DATA_BLOCK "_2010SC130U01TSH01_DB"   // DB2038
TITLE = Instance DB Alarm: Break Resistor Temp High
{ S7_Optimized_Access := 'FALSE' }
AUTHOR : 7Art
NAME : ALARM_DB
VERSION : 8.0
// stored: InstanceOfName ACESYS_ALARM
"ACESYS_ALARM"
BEGIN
   FP_PARM.EnableTime_Low_Pre := 5;
   FP_EN.Alarm_Low := TRUE;
   PWR := TRUE;
   EN_L := TRUE;
   OK := TRUE;
   AL_L := TRUE;
   AL_H := TRUE;
   WARN_L := TRUE;
   WARN_H := TRUE;
   MSW.EXT.Operation := TRUE;
   MSW.Status := 2;
   MSW.TimeStamp := 16#7ECD;
   BlockInfo.Ace_Version := 80;
   BlockInfo.Ace_BuildNo := 4;
   BlockInfo.State_Act := 2;
   BlockInfo.State_Prev := 202;
   BlockInfo.DB_Number := 2038;
   FP_PARM.EnableTime_Low_Acc := 5;
   FP_SIM.SIG_Enable := TRUE;
   FP_SIM.PWR_Enable := TRUE;
   ONS.SecPulse1 := TRUE;
   ONS.AL_L_Aux := TRUE;
   ONS.AL_H_Aux := TRUE;
   EnableTime_Low_Done := TRUE;
   StatusWork := 2;
   OUT.OK := TRUE;
   OUT.AL_L := TRUE;
   OUT.AL_H := TRUE;
   OUT.WARN_L := TRUE;
   OUT.WARN_H := TRUE;
   MSW_Status_Trans := 2;
END_DATA_BLOCK

DATA_BLOCK "_2010CR150M01OAC01_DB"   // DB2039
TITLE = Instance DB Alarm: Emergency stop PB
{ S7_Optimized_Access := 'FALSE' }
AUTHOR : 7Art
NAME : ALARM_DB
VERSION : 8.0
// stored: InstanceOfName ACESYS_ALARM
"ACESYS_ALARM"
BEGIN
   FP_PARM.EnableTime_Low_Pre := 5;
   FP_EN.Alarm_Low := TRUE;
   PWR := TRUE;
   EN_L := TRUE;
   OK := TRUE;
   AL_L := TRUE;
   AL_H := TRUE;
   WARN_L := TRUE;
   WARN_H := TRUE;
   MSW.EXT.Operation := TRUE;
   MSW.Status := 2;
   MSW.TimeStamp := 16#72EA;
   BlockInfo.Ace_Version := 80;
   BlockInfo.Ace_BuildNo := 4;
   BlockInfo.State_Act := 2;
   BlockInfo.State_Prev := 202;
   BlockInfo.DB_Number := 2039;
   FP_PARM.EnableTime_Low_Acc := 5;
   FP_SIM.SIG_Enable := TRUE;
   FP_SIM.PWR_Enable := TRUE;
   ONS.SecPulse1 := TRUE;
   ONS.AL_L_Aux := TRUE;
   ONS.AL_H_Aux := TRUE;
   EnableTime_Low_Done := TRUE;
   StatusWork := 2;
   OUT.OK := TRUE;
   OUT.AL_L := TRUE;
   OUT.AL_H := TRUE;
   OUT.WARN_L := TRUE;
   OUT.WARN_H := TRUE;
   MSW_Status_Trans := 2;
END_DATA_BLOCK

DATA_BLOCK "_2010CR150M01YSQ01_DB"   // DB2040
TITLE = Instance DB Alarm: Breaker feedback
{ S7_Optimized_Access := 'FALSE' }
AUTHOR : 7Art
NAME : ALARM_DB
VERSION : 8.0
// stored: InstanceOfName ACESYS_ALARM
"ACESYS_ALARM"
BEGIN
   FP_PARM.EnableTime_Low_Pre := 5;
   FP_EN.Alarm_Low := TRUE;
   PWR := TRUE;
   EN_L := TRUE;
   OK := TRUE;
   AL_L := TRUE;
   AL_H := TRUE;
   WARN_L := TRUE;
   WARN_H := TRUE;
   MSW.EXT.Operation := TRUE;
   MSW.Status := 2;
   MSW.TimeStamp := 16#8D11;
   BlockInfo.Ace_Version := 80;
   BlockInfo.Ace_BuildNo := 4;
   BlockInfo.State_Act := 2;
   BlockInfo.State_Prev := 202;
   BlockInfo.DB_Number := 2040;
   FP_PARM.EnableTime_Low_Acc := 5;
   FP_SIM.SIG_Enable := TRUE;
   FP_SIM.PWR_Enable := TRUE;
   ONS.SecPulse1 := TRUE;
   ONS.AL_L_Aux := TRUE;
   ONS.AL_H_Aux := TRUE;
   EnableTime_Low_Done := TRUE;
   StatusWork := 2;
   OUT.OK := TRUE;
   OUT.AL_L := TRUE;
   OUT.AL_H := TRUE;
   OUT.WARN_L := TRUE;
   OUT.WARN_H := TRUE;
   MSW_Status_Trans := 2;
END_DATA_BLOCK

DATA_BLOCK "_2010CR150M01NS01_DB"   // DB2041
TITLE = Instance DB Alarm: PTS Sensor
{ S7_Optimized_Access := 'FALSE' }
AUTHOR : 7Art
NAME : ALARM_DB
VERSION : 8.0
// stored: InstanceOfName ACESYS_ALARM
"ACESYS_ALARM"
BEGIN
   FP_PARM.EnableTime_Low_Pre := 5;
   FP_EN.Alarm_Low := TRUE;
   PWR := TRUE;
   EN_L := TRUE;
   OK := TRUE;
   AL_L := TRUE;
   AL_H := TRUE;
   WARN_L := TRUE;
   WARN_H := TRUE;
   MSW.EXT.Operation := TRUE;
   MSW.Status := 2;
   MSW.TimeStamp := 16#08E4;
   BlockInfo.Ace_Version := 80;
   BlockInfo.Ace_BuildNo := 4;
   BlockInfo.State_Act := 2;
   BlockInfo.State_Prev := 202;
   BlockInfo.DB_Number := 2041;
   FP_PARM.EnableTime_Low_Acc := 5;
   FP_SIM.SIG_Enable := TRUE;
   FP_SIM.PWR_Enable := TRUE;
   ONS.SecPulse1 := TRUE;
   ONS.AL_L_Aux := TRUE;
   ONS.AL_H_Aux := TRUE;
   EnableTime_Low_Done := TRUE;
   StatusWork := 2;
   OUT.OK := TRUE;
   OUT.AL_L := TRUE;
   OUT.AL_H := TRUE;
   OUT.WARN_L := TRUE;
   OUT.WARN_H := TRUE;
   MSW_Status_Trans := 2;
END_DATA_BLOCK

DATA_BLOCK "_2010PMC01YSH01_DB"   // DB2042
TITLE = Instance DB Alarm: PTS Sensor
{ S7_Optimized_Access := 'FALSE' }
AUTHOR : 7Art
NAME : ALARM_DB
VERSION : 8.0
// stored: InstanceOfName ACESYS_ALARM
"ACESYS_ALARM"
BEGIN
   FP_PARM.EnableTime_Low_Pre := 5;
   FP_EN.Alarm_Low := TRUE;
   PWR := TRUE;
   EN_L := TRUE;
   OK := TRUE;
   AL_L := TRUE;
   AL_H := TRUE;
   WARN_L := TRUE;
   WARN_H := TRUE;
   MSW.EXT.Operation := TRUE;
   MSW.Status := 2;
   MSW.TimeStamp := 16#8C12;
   BlockInfo.Ace_Version := 80;
   BlockInfo.Ace_BuildNo := 4;
   BlockInfo.State_Act := 2;
   BlockInfo.State_Prev := 202;
   BlockInfo.DB_Number := 2042;
   FP_PARM.EnableTime_Low_Acc := 5;
   FP_SIM.SIG_Enable := TRUE;
   FP_SIM.PWR_Enable := TRUE;
   ONS.SecPulse1 := TRUE;
   ONS.AL_L_Aux := TRUE;
   ONS.AL_H_Aux := TRUE;
   EnableTime_Low_Done := TRUE;
   StatusWork := 2;
   OUT.OK := TRUE;
   OUT.AL_L := TRUE;
   OUT.AL_H := TRUE;
   OUT.WARN_L := TRUE;
   OUT.WARN_H := TRUE;
   MSW_Status_Trans := 2;
END_DATA_BLOCK

DATA_BLOCK "_2010PMC01YSQ10G01_DB"   // DB2043
TITLE = Instance DB Alarm: PTS Sensor
{ S7_Optimized_Access := 'FALSE' }
AUTHOR : 7Art
NAME : ALARM_DB
VERSION : 8.0
// stored: InstanceOfName ACESYS_ALARM
"ACESYS_ALARM"
BEGIN
   FP_PARM.EnableTime_Low_Pre := 5;
   FP_EN.Alarm_Low := TRUE;
   PWR := TRUE;
   EN_L := TRUE;
   OK := TRUE;
   AL_L := TRUE;
   AL_H := TRUE;
   WARN_L := TRUE;
   WARN_H := TRUE;
   MSW.EXT.Operation := TRUE;
   MSW.Status := 2;
   MSW.TimeStamp := 16#8BF2;
   BlockInfo.Ace_Version := 80;
   BlockInfo.Ace_BuildNo := 4;
   BlockInfo.State_Act := 2;
   BlockInfo.State_Prev := 202;
   BlockInfo.DB_Number := 2043;
   FP_PARM.EnableTime_Low_Acc := 5;
   FP_SIM.SIG_Enable := TRUE;
   FP_SIM.PWR_Enable := TRUE;
   ONS.SecPulse2 := TRUE;
   ONS.AL_L_Aux := TRUE;
   ONS.AL_H_Aux := TRUE;
   EnableTime_Low_Done := TRUE;
   Sec_Pulse := TRUE;
   StatusWork := 2;
   OUT.OK := TRUE;
   OUT.AL_L := TRUE;
   OUT.AL_H := TRUE;
   OUT.WARN_L := TRUE;
   OUT.WARN_H := TRUE;
   MSW_Status_Trans := 2;
END_DATA_BLOCK

DATA_BLOCK "_2010PMC01YSQ10Q03_DB"   // DB2044
TITLE = Instance DB Alarm: PTS Sensor
{ S7_Optimized_Access := 'FALSE' }
AUTHOR : 7Art
NAME : ALARM_DB
VERSION : 8.0
// stored: InstanceOfName ACESYS_ALARM
"ACESYS_ALARM"
BEGIN
   FP_PARM.EnableTime_Low_Pre := 5;
   FP_EN.Alarm_Low := TRUE;
   PWR := TRUE;
   EN_L := TRUE;
   OK := TRUE;
   AL_L := TRUE;
   AL_H := TRUE;
   WARN_L := TRUE;
   WARN_H := TRUE;
   MSW.EXT.Operation := TRUE;
   MSW.Status := 2;
   MSW.TimeStamp := 16#7EC5;
   BlockInfo.Ace_Version := 80;
   BlockInfo.Ace_BuildNo := 4;
   BlockInfo.State_Act := 2;
   BlockInfo.State_Prev := 202;
   BlockInfo.DB_Number := 2044;
   FP_PARM.EnableTime_Low_Acc := 5;
   FP_SIM.SIG_Enable := TRUE;
   FP_SIM.PWR_Enable := TRUE;
   ONS.SecPulse2 := TRUE;
   ONS.AL_L_Aux := TRUE;
   ONS.AL_H_Aux := TRUE;
   EnableTime_Low_Done := TRUE;
   Sec_Pulse := TRUE;
   StatusWork := 2;
   OUT.OK := TRUE;
   OUT.AL_L := TRUE;
   OUT.AL_H := TRUE;
   OUT.WARN_L := TRUE;
   OUT.WARN_H := TRUE;
   MSW_Status_Trans := 2;
END_DATA_BLOCK

DATA_BLOCK "_2010PMC01YSQ20Q03_DB"   // DB2045
TITLE = Instance DB Alarm: PTS Sensor
{ S7_Optimized_Access := 'FALSE' }
AUTHOR : 7Art
NAME : ALARM_DB
VERSION : 8.0
// stored: InstanceOfName ACESYS_ALARM
"ACESYS_ALARM"
BEGIN
   FP_PARM.EnableTime_Low_Pre := 5;
   FP_EN.Alarm_Low := TRUE;
   PWR := TRUE;
   EN_L := TRUE;
   OK := TRUE;
   AL_L := TRUE;
   AL_H := TRUE;
   WARN_L := TRUE;
   WARN_H := TRUE;
   MSW.EXT.Operation := TRUE;
   MSW.Status := 2;
   MSW.TimeStamp := 16#72EA;
   BlockInfo.Ace_Version := 80;
   BlockInfo.Ace_BuildNo := 4;
   BlockInfo.State_Act := 2;
   BlockInfo.State_Prev := 202;
   BlockInfo.DB_Number := 2045;
   FP_PARM.EnableTime_Low_Acc := 5;
   FP_SIM.SIG_Enable := TRUE;
   FP_SIM.PWR_Enable := TRUE;
   ONS.SecPulse2 := TRUE;
   ONS.AL_L_Aux := TRUE;
   ONS.AL_H_Aux := TRUE;
   EnableTime_Low_Done := TRUE;
   StatusWork := 2;
   OUT.OK := TRUE;
   OUT.AL_L := TRUE;
   OUT.AL_H := TRUE;
   OUT.WARN_L := TRUE;
   OUT.WARN_H := TRUE;
   MSW_Status_Trans := 2;
END_DATA_BLOCK

DATA_BLOCK "_2010PMC01YSQ20Q04_DB"   // DB2046
TITLE = Instance DB Alarm: PTS Sensor
{ S7_Optimized_Access := 'FALSE' }
AUTHOR : 7Art
NAME : ALARM_DB
VERSION : 8.0
// stored: InstanceOfName ACESYS_ALARM
"ACESYS_ALARM"
BEGIN
   FP_PARM.EnableTime_Low_Pre := 5;
   FP_EN.Alarm_Low := TRUE;
   PWR := TRUE;
   EN_L := TRUE;
   OK := TRUE;
   AL_L := TRUE;
   AL_H := TRUE;
   WARN_L := TRUE;
   WARN_H := TRUE;
   MSW.EXT.Operation := TRUE;
   MSW.Status := 2;
   MSW.TimeStamp := 16#72EA;
   BlockInfo.Ace_Version := 80;
   BlockInfo.Ace_BuildNo := 4;
   BlockInfo.State_Act := 2;
   BlockInfo.State_Prev := 202;
   BlockInfo.DB_Number := 2046;
   FP_PARM.EnableTime_Low_Acc := 5;
   FP_SIM.SIG_Enable := TRUE;
   FP_SIM.PWR_Enable := TRUE;
   ONS.SecPulse2 := TRUE;
   ONS.AL_L_Aux := TRUE;
   ONS.AL_H_Aux := TRUE;
   EnableTime_Low_Done := TRUE;
   StatusWork := 2;
   OUT.OK := TRUE;
   OUT.AL_L := TRUE;
   OUT.AL_H := TRUE;
   OUT.WARN_L := TRUE;
   OUT.WARN_H := TRUE;
   MSW_Status_Trans := 2;
END_DATA_BLOCK

DATA_BLOCK "_2010PMC01YSQ26Q01_DB"   // DB2047
TITLE = Instance DB Alarm: PTS Sensor
{ S7_Optimized_Access := 'FALSE' }
AUTHOR : 7Art
NAME : ALARM_DB
VERSION : 8.0
// stored: InstanceOfName ACESYS_ALARM
"ACESYS_ALARM"
BEGIN
   FP_PARM.EnableTime_Low_Pre := 5;
   FP_EN.Alarm_Low := TRUE;
   PWR := TRUE;
   EN_L := TRUE;
   OK := TRUE;
   AL_L := TRUE;
   AL_H := TRUE;
   WARN_L := TRUE;
   WARN_H := TRUE;
   MSW.EXT.Operation := TRUE;
   MSW.Status := 2;
   MSW.TimeStamp := 16#61B4;
   BlockInfo.Ace_Version := 80;
   BlockInfo.Ace_BuildNo := 4;
   BlockInfo.State_Act := 2;
   BlockInfo.State_Prev := 202;
   BlockInfo.DB_Number := 2047;
   FP_PARM.EnableTime_Low_Acc := 5;
   FP_SIM.SIG_Enable := TRUE;
   FP_SIM.PWR_Enable := TRUE;
   ONS.SecPulse2 := TRUE;
   ONS.AL_L_Aux := TRUE;
   ONS.AL_H_Aux := TRUE;
   EnableTime_Low_Done := TRUE;
   StatusWork := 2;
   OUT.OK := TRUE;
   OUT.AL_L := TRUE;
   OUT.AL_H := TRUE;
   OUT.WARN_L := TRUE;
   OUT.WARN_H := TRUE;
   MSW_Status_Trans := 2;
END_DATA_BLOCK

DATA_BLOCK "_2010PMC01YSQ30Q02_DB"   // DB2048
TITLE = Instance DB Alarm: PTS Sensor
{ S7_Optimized_Access := 'FALSE' }
AUTHOR : 7Art
NAME : ALARM_DB
VERSION : 8.0
// stored: InstanceOfName ACESYS_ALARM
"ACESYS_ALARM"
BEGIN
   FP_PARM.EnableTime_Low_Pre := 5;
   FP_EN.Alarm_Low := TRUE;
   PWR := TRUE;
   EN_L := TRUE;
   OK := TRUE;
   AL_L := TRUE;
   AL_H := TRUE;
   WARN_L := TRUE;
   WARN_H := TRUE;
   MSW.EXT.Operation := TRUE;
   MSW.EXT.Forced := TRUE;
   MSW.Status := 2;
   MSW.TimeStamp := 16#166B;
   BlockInfo.Ace_Version := 80;
   BlockInfo.Ace_BuildNo := 4;
   BlockInfo.State_Act := 2;
   BlockInfo.State_Prev := 1;
   BlockInfo.DB_Number := 2048;
   FP_SEL.Force_OK := TRUE;
   FP_PARM.EnableTime_Low_Acc := 5;
   FP_SIM.SIG_Enable := TRUE;
   FP_SIM.PWR_Enable := TRUE;
   ONS.ForceOK := TRUE;
   ONS.SecPulse2 := TRUE;
   ONS.AL_L_Aux := TRUE;
   ONS.AL_H_Aux := TRUE;
   EnableTime_Low_Done := TRUE;
   StatusWork := 2;
   OUT.OK := TRUE;
   OUT.AL_L := TRUE;
   OUT.AL_H := TRUE;
   OUT.WARN_L := TRUE;
   OUT.WARN_H := TRUE;
   MSW_Status_Trans := 2;
END_DATA_BLOCK

DATA_BLOCK "_2010PMC01YSQ30Q03_DB"   // DB2049
TITLE = Instance DB Alarm: PTS Sensor
{ S7_Optimized_Access := 'FALSE' }
AUTHOR : 7Art
NAME : ALARM_DB
VERSION : 8.0
// stored: InstanceOfName ACESYS_ALARM
"ACESYS_ALARM"
BEGIN
   FP_PARM.EnableTime_Low_Pre := 5;
   FP_EN.Alarm_Low := TRUE;
   PWR := TRUE;
   EN_L := TRUE;
   OK := TRUE;
   AL_L := TRUE;
   AL_H := TRUE;
   WARN_L := TRUE;
   WARN_H := TRUE;
   MSW.EXT.Operation := TRUE;
   MSW.Status := 2;
   MSW.TimeStamp := 16#72EA;
   BlockInfo.Ace_Version := 80;
   BlockInfo.Ace_BuildNo := 4;
   BlockInfo.State_Act := 2;
   BlockInfo.State_Prev := 202;
   BlockInfo.DB_Number := 2049;
   FP_PARM.EnableTime_Low_Acc := 5;
   FP_SIM.SIG_Enable := TRUE;
   FP_SIM.PWR_Enable := TRUE;
   ONS.SecPulse2 := TRUE;
   ONS.AL_L_Aux := TRUE;
   ONS.AL_H_Aux := TRUE;
   EnableTime_Low_Done := TRUE;
   StatusWork := 2;
   OUT.OK := TRUE;
   OUT.AL_L := TRUE;
   OUT.AL_H := TRUE;
   OUT.WARN_L := TRUE;
   OUT.WARN_H := TRUE;
   MSW_Status_Trans := 2;
END_DATA_BLOCK

DATA_BLOCK "_2010PMC01UPS01_DB"   // DB2050
TITLE = Instance DB Alarm: PTS Sensor
{ S7_Optimized_Access := 'FALSE' }
AUTHOR : 7Art
NAME : ALARM_DB
VERSION : 8.0
// stored: InstanceOfName ACESYS_ALARM
"ACESYS_ALARM"
BEGIN
   FP_PARM.EnableTime_Low_Pre := 5;
   FP_EN.Alarm_Low := TRUE;
   SIG := FALSE;
   PWR := TRUE;
   EN_L := TRUE;
   OK := TRUE;
   AL_L := TRUE;
   AL_H := TRUE;
   WARN_L := TRUE;
   WARN_H := TRUE;
   MSW.EXT.Operation := TRUE;
   MSW.EXT.Forced := TRUE;
   MSW.Status := 1;
   MSW.TimeStamp := 16#AFF4;
   BlockInfo.Ace_Version := 80;
   BlockInfo.Ace_BuildNo := 4;
   BlockInfo.State_Act := 1;
   BlockInfo.State_Prev := 2;
   BlockInfo.DB_Number := 2050;
   FP_SEL.Force_OK := TRUE;
   FP_PARM.EnableTime_Low_Acc := 5;
   FP_SIM.SIG_Enable := TRUE;
   FP_SIM.PWR_Enable := TRUE;
   ONS.ForceOK := TRUE;
   ONS.SecPulse2 := TRUE;
   ONS.AL_L_Aux := TRUE;
   ONS.AL_H_Aux := TRUE;
   EnableTime_Low_Done := TRUE;
   AlarmDelay_Low_Done := TRUE;
   StatusWork := 1;
   OUT.OK := TRUE;
   OUT.AL_L := TRUE;
   OUT.AL_H := TRUE;
   OUT.WARN_L := TRUE;
   OUT.WARN_H := TRUE;
   MSW_Status_Trans := 1;
END_DATA_BLOCK

DATA_BLOCK "_2010PMC01OA03_DB"   // DB2051
TITLE = Instance DB Alarm: PTS Sensor
{ S7_Optimized_Access := 'FALSE' }
AUTHOR : 7Art
NAME : ALARM_DB
VERSION : 8.0
// stored: InstanceOfName ACESYS_ALARM
"ACESYS_ALARM"
BEGIN
   FP_PARM.EnableTime_Low_Pre := 5;
   FP_EN.Alarm_Low := TRUE;
   PWR := TRUE;
   EN_L := TRUE;
   OK := TRUE;
   AL_L := TRUE;
   AL_H := TRUE;
   WARN_L := TRUE;
   WARN_H := TRUE;
   MSW.EXT.Operation := TRUE;
   MSW.Status := 2;
   MSW.TimeStamp := 16#B81A;
   BlockInfo.Ace_Version := 80;
   BlockInfo.Ace_BuildNo := 4;
   BlockInfo.State_Act := 2;
   BlockInfo.State_Prev := 202;
   BlockInfo.DB_Number := 2051;
   FP_PARM.EnableTime_Low_Acc := 5;
   FP_SIM.SIG_Enable := TRUE;
   FP_SIM.PWR_Enable := TRUE;
   ONS.SecPulse2 := TRUE;
   ONS.AL_L_Aux := TRUE;
   ONS.AL_H_Aux := TRUE;
   EnableTime_Low_Done := TRUE;
   StatusWork := 2;
   OUT.OK := TRUE;
   OUT.AL_L := TRUE;
   OUT.AL_H := TRUE;
   OUT.WARN_L := TRUE;
   OUT.WARN_H := TRUE;
   MSW_Status_Trans := 2;
END_DATA_BLOCK

DATA_BLOCK "_2010PMC01YSES50FES01_DB"   // DB2052
TITLE = Instance DB Alarm: PTS Sensor
{ S7_Optimized_Access := 'FALSE' }
AUTHOR : 7Art
NAME : ALARM_DB
VERSION : 8.0
// stored: InstanceOfName ACESYS_ALARM
"ACESYS_ALARM"
BEGIN
   FP_PARM.EnableTime_Low_Pre := 5;
   FP_EN.Alarm_Low := TRUE;
   PWR := TRUE;
   EN_L := TRUE;
   OK := TRUE;
   AL_L := TRUE;
   AL_H := TRUE;
   WARN_L := TRUE;
   WARN_H := TRUE;
   MSW.EXT.Operation := TRUE;
   MSW.Status := 2;
   MSW.TimeStamp := 16#A4ED;
   BlockInfo.Ace_Version := 80;
   BlockInfo.Ace_BuildNo := 4;
   BlockInfo.State_Act := 2;
   BlockInfo.State_Prev := 202;
   BlockInfo.DB_Number := 2052;
   FP_PARM.EnableTime_Low_Acc := 5;
   FP_SIM.SIG_Enable := TRUE;
   FP_SIM.PWR_Enable := TRUE;
   ONS.SecPulse2 := TRUE;
   ONS.AL_L_Aux := TRUE;
   ONS.AL_H_Aux := TRUE;
   EnableTime_Low_Done := TRUE;
   StatusWork := 2;
   OUT.OK := TRUE;
   OUT.AL_L := TRUE;
   OUT.AL_H := TRUE;
   OUT.WARN_L := TRUE;
   OUT.WARN_H := TRUE;
   MSW_Status_Trans := 2;
END_DATA_BLOCK

DATA_BLOCK "_2010PMC01OA01_DB"   // DB2053
TITLE = Instance DB Alarm: PTS Sensor
{ S7_Optimized_Access := 'FALSE' }
AUTHOR : 7Art
NAME : ALARM_DB
VERSION : 8.0
// stored: InstanceOfName ACESYS_ALARM
"ACESYS_ALARM"
BEGIN
   FP_PARM.EnableTime_Low_Pre := 5;
   FP_EN.Alarm_Low := TRUE;
   PWR := TRUE;
   EN_L := TRUE;
   OK := TRUE;
   AL_L := TRUE;
   AL_H := TRUE;
   WARN_L := TRUE;
   WARN_H := TRUE;
   MSW.EXT.Operation := TRUE;
   MSW.Status := 2;
   MSW.TimeStamp := 16#7EC5;
   BlockInfo.Ace_Version := 80;
   BlockInfo.Ace_BuildNo := 4;
   BlockInfo.State_Act := 2;
   BlockInfo.State_Prev := 202;
   BlockInfo.DB_Number := 2053;
   FP_PARM.EnableTime_Low_Acc := 5;
   FP_SIM.SIG_Enable := TRUE;
   FP_SIM.PWR_Enable := TRUE;
   ONS.SecPulse2 := TRUE;
   ONS.AL_L_Aux := TRUE;
   ONS.AL_H_Aux := TRUE;
   EnableTime_Low_Done := TRUE;
   StatusWork := 2;
   OUT.OK := TRUE;
   OUT.AL_L := TRUE;
   OUT.AL_H := TRUE;
   OUT.WARN_L := TRUE;
   OUT.WARN_H := TRUE;
   MSW_Status_Trans := 2;
END_DATA_BLOCK

DATA_BLOCK "_2010BF110YSQ02_DB"   // DB2054
TITLE = Instance DB Alarm: PTS Sensor
{ S7_Optimized_Access := 'FALSE' }
AUTHOR : 7Art
NAME : ALARM_DB
VERSION : 8.0
// stored: InstanceOfName ACESYS_ALARM
"ACESYS_ALARM"
BEGIN
   FP_PARM.EnableTime_Low_Pre := 5;
   FP_EN.Alarm_Low := TRUE;
   SIG := FALSE;
   PWR := TRUE;
   EN_L := TRUE;
   OK := TRUE;
   AL_L := TRUE;
   AL_H := TRUE;
   WARN_L := TRUE;
   WARN_H := TRUE;
   MSW.EXT.Operation := TRUE;
   MSW.EXT.Forced := TRUE;
   MSW.Status := 1;
   MSW.TimeStamp := 16#AC7B;
   BlockInfo.Ace_Version := 80;
   BlockInfo.Ace_BuildNo := 4;
   BlockInfo.State_Act := 1;
   BlockInfo.State_Prev := 202;
   BlockInfo.DB_Number := 2054;
   FP_SEL.Force_OK := TRUE;
   FP_PARM.EnableTime_Low_Acc := 5;
   FP_SIM.SIG_Enable := TRUE;
   FP_SIM.PWR_Enable := TRUE;
   ONS.ForceOK := TRUE;
   ONS.SecPulse2 := TRUE;
   ONS.AL_L_Aux := TRUE;
   ONS.AL_H_Aux := TRUE;
   EnableTime_Low_Done := TRUE;
   AlarmDelay_Low_Done := TRUE;
   StatusWork := 1;
   OUT.OK := TRUE;
   OUT.AL_L := TRUE;
   OUT.AL_H := TRUE;
   OUT.WARN_L := TRUE;
   OUT.WARN_H := TRUE;
   MSW_Status_Trans := 1;
END_DATA_BLOCK

DATA_BLOCK "_2010PMC01PS01_DB"   // DB2055
TITLE = Instance DB Alarm: PTS Sensor
{ S7_Optimized_Access := 'FALSE' }
AUTHOR : 7Art
NAME : ALARM_DB
VERSION : 8.0
// stored: InstanceOfName ACESYS_ALARM
"ACESYS_ALARM"
BEGIN
   FP_PARM.EnableTime_Low_Pre := 5;
   FP_EN.Alarm_Low := TRUE;
   PWR := TRUE;
   EN_L := TRUE;
   OK := TRUE;
   AL_L := TRUE;
   AL_H := TRUE;
   WARN_L := TRUE;
   WARN_H := TRUE;
   MSW.EXT.Operation := TRUE;
   MSW.Status := 2;
   MSW.TimeStamp := 16#8C12;
   BlockInfo.Ace_Version := 80;
   BlockInfo.Ace_BuildNo := 4;
   BlockInfo.State_Act := 2;
   BlockInfo.State_Prev := 202;
   BlockInfo.DB_Number := 2055;
   FP_PARM.EnableTime_Low_Acc := 5;
   FP_SIM.SIG_Enable := TRUE;
   FP_SIM.PWR_Enable := TRUE;
   ONS.SecPulse2 := TRUE;
   ONS.AL_L_Aux := TRUE;
   ONS.AL_H_Aux := TRUE;
   EnableTime_Low_Done := TRUE;
   StatusWork := 2;
   OUT.OK := TRUE;
   OUT.AL_L := TRUE;
   OUT.AL_H := TRUE;
   OUT.WARN_L := TRUE;
   OUT.WARN_H := TRUE;
   MSW_Status_Trans := 2;
END_DATA_BLOCK

DATA_BLOCK "_2010PMC01YSH01_DB_15"   // DB2056
TITLE = Instance DB Alarm: PTS Sensor
{ S7_Optimized_Access := 'FALSE' }
AUTHOR : 7Art
NAME : ALARM_DB
VERSION : 8.0
// stored: InstanceOfName ACESYS_ALARM
"ACESYS_ALARM"
BEGIN
   FP_PARM.EnableTime_Low_Pre := 5;
   FP_EN.ParentSupress := TRUE;
   FP_EN.ParentSupressUnit := TRUE;
   FP_EN.Alarm_Low := TRUE;
   SIG := FALSE;
   PWR := TRUE;
   EN_L := TRUE;
   AL_H := TRUE;
   WARN_L := TRUE;
   WARN_H := TRUE;
   MSW.EXT.AlarmPresent := TRUE;
   MSW.EXT.AlarmFailUnAck := TRUE;
   MSW.Status := 202;
   MSW.TimeStamp := 16#60BB;
   BlockInfo.Ace_Version := 80;
   BlockInfo.Ace_BuildNo := 4;
   BlockInfo.State_Act := 202;
   BlockInfo.State_Prev := 1;
   BlockInfo.DB_Number := 2000;
   FP_PARM.EnableTime_Low_Acc := 5;
   FP_SIM.SIG_Enable := TRUE;
   FP_SIM.PWR_Enable := TRUE;
   ONS.SecPulse2 := TRUE;
   ONS.ALARM_AlarmCondition := TRUE;
   ONS.AL_H_Aux := TRUE;
   EnableTime_Low_Done := TRUE;
   AlarmDelay_Low_Done := TRUE;
   ALARM_AlarmPresent := TRUE;
   StatusWork := 202;
   AlarmNo := 4;
   AlarmNo_Old := 4;
   OUT.AL_H := TRUE;
   OUT.WARN_L := TRUE;
   OUT.WARN_H := TRUE;
   MSW_EXT_AlarmFailUnAck := TRUE;
   MSW_Status_Trans := 202;
END_DATA_BLOCK

DATA_BLOCK "_2010PMC01YSQ42Q02"   // DB2057
TITLE = Instance DB Alarm: PTS Sensor
{ S7_Optimized_Access := 'FALSE' }
AUTHOR : 7Art
NAME : ALARM_DB
VERSION : 8.0
// stored: InstanceOfName ACESYS_ALARM
"ACESYS_ALARM"
BEGIN
   FP_PARM.EnableTime_Low_Pre := 5;
   FP_EN.Alarm_Low := TRUE;
   PWR := TRUE;
   EN_L := TRUE;
   OK := TRUE;
   AL_L := TRUE;
   AL_H := TRUE;
   WARN_L := TRUE;
   WARN_H := TRUE;
   MSW.EXT.Operation := TRUE;
   MSW.Status := 2;
   MSW.TimeStamp := 16#72EA;
   BlockInfo.Ace_Version := 80;
   BlockInfo.Ace_BuildNo := 4;
   BlockInfo.State_Act := 2;
   BlockInfo.State_Prev := 202;
   BlockInfo.DB_Number := 2057;
   FP_PARM.EnableTime_Low_Acc := 5;
   FP_SIM.SIG_Enable := TRUE;
   FP_SIM.PWR_Enable := TRUE;
   ONS.SecPulse2 := TRUE;
   ONS.AL_L_Aux := TRUE;
   ONS.AL_H_Aux := TRUE;
   EnableTime_Low_Done := TRUE;
   StatusWork := 2;
   OUT.OK := TRUE;
   OUT.AL_L := TRUE;
   OUT.AL_H := TRUE;
   OUT.WARN_L := TRUE;
   OUT.WARN_H := TRUE;
   MSW_Status_Trans := 2;
END_DATA_BLOCK

DATA_BLOCK "_2010CV180GC01_DB"   // DB2058
TITLE = Instance DB Alarm: _2010CV180OAC01
{ S7_Optimized_Access := 'FALSE' }
AUTHOR : METIS
NAME : ALARM_DB
VERSION : 8.0
// stored: InstanceOfName ACESYS_ALARM
"ACESYS_ALARM"
BEGIN
   FP_PARM.EnableTime_Low_Pre := 5;
   FP_EN.Alarm_Low := TRUE;
   PWR := TRUE;
   EN_L := TRUE;
   OK := TRUE;
   AL_L := TRUE;
   AL_H := TRUE;
   WARN_L := TRUE;
   WARN_H := TRUE;
   MSW.EXT.Operation := TRUE;
   MSW.Status := 2;
   MSW.TimeStamp := 16#3365;
   BlockInfo.Ace_Version := 80;
   BlockInfo.Ace_BuildNo := 4;
   BlockInfo.State_Act := 2;
   BlockInfo.State_Prev := 1;
   BlockInfo.DB_Number := 2058;
   FP_PARM.EnableTime_Low_Acc := 5;
   FP_SIM.SIG_Enable := TRUE;
   FP_SIM.PWR_Enable := TRUE;
   ONS.SecPulse2 := TRUE;
   ONS.AL_L_Aux := TRUE;
   ONS.AL_H_Aux := TRUE;
   EnableTime_Low_Done := TRUE;
   StatusWork := 2;
   OUT.OK := TRUE;
   OUT.AL_L := TRUE;
   OUT.AL_H := TRUE;
   OUT.WARN_L := TRUE;
   OUT.WARN_H := TRUE;
   MSW_Status_Trans := 2;
END_DATA_BLOCK

DATA_BLOCK "_2010CV120GC01_DB"   // DB2059
TITLE = Instance DB Alarm: _2010CV180OAC01
{ S7_Optimized_Access := 'FALSE' }
AUTHOR : METIS
NAME : ALARM_DB
VERSION : 8.0
// stored: InstanceOfName ACESYS_ALARM
"ACESYS_ALARM"
BEGIN
   FP_PARM.EnableTime_Low_Pre := 5;
   FP_EN.Alarm_Low := TRUE;
   PWR := TRUE;
   EN_L := TRUE;
   OK := TRUE;
   AL_L := TRUE;
   AL_H := TRUE;
   WARN_L := TRUE;
   WARN_H := TRUE;
   MSW.EXT.Operation := TRUE;
   MSW.Status := 2;
   MSW.TimeStamp := 16#36C9;
   BlockInfo.Ace_Version := 80;
   BlockInfo.Ace_BuildNo := 4;
   BlockInfo.State_Act := 2;
   BlockInfo.State_Prev := 1;
   BlockInfo.DB_Number := 2059;
   FP_PARM.EnableTime_Low_Acc := 5;
   FP_SIM.SIG_Enable := TRUE;
   FP_SIM.PWR_Enable := TRUE;
   ONS.SecPulse2 := TRUE;
   ONS.AL_L_Aux := TRUE;
   ONS.AL_H_Aux := TRUE;
   EnableTime_Low_Done := TRUE;
   StatusWork := 2;
   OUT.OK := TRUE;
   OUT.AL_L := TRUE;
   OUT.AL_H := TRUE;
   OUT.WARN_L := TRUE;
   OUT.WARN_H := TRUE;
   MSW_Status_Trans := 2;
END_DATA_BLOCK

DATA_BLOCK "_2010SJ950D01L41_DB"   // DB2121
TITLE = Instance DB Alarm: _2010SJ950D01L41
{ S7_Optimized_Access := 'FALSE' }
AUTHOR : METIS
NAME : ALARM_DB
VERSION : 8.0
// stored: InstanceOfName ACESYS_ALARM
"ACESYS_ALARM"
BEGIN
   FP_PARM.EnableTime_Low_Pre := 5;
   FP_EN.ParentSupress := TRUE;
   FP_EN.ParentSupressUnit := TRUE;
   FP_EN.Alarm_Low := TRUE;
   SIG := FALSE;
   PWR := TRUE;
   EN_L := TRUE;
   AL_SUPR := TRUE;
   AL_H := TRUE;
   WARN_L := TRUE;
   WARN_H := TRUE;
   MSW.EXT.AlarmSuppressed := TRUE;
   MSW.EXT.AlarmPresent := TRUE;
   MSW.EXT.AlarmFailUnAck := TRUE;
   MSW.Status := 202;
   MSW.TimeStamp := 16#524E;
   BlockInfo.Ace_Version := 80;
   BlockInfo.Ace_BuildNo := 4;
   BlockInfo.State_Act := 202;
   BlockInfo.State_Prev := 1;
   BlockInfo.DB_Number := 2121;
   FP_PARM.EnableTime_Low_Acc := 5;
   FP_SIM.SIG_Enable := TRUE;
   FP_SIM.PWR_Enable := TRUE;
   ONS.SecPulse2 := TRUE;
   ONS.ALARM_AlarmCondition := TRUE;
   ONS.AL_H_Aux := TRUE;
   EnableTime_Low_Done := TRUE;
   AlarmDelay_Low_Done := TRUE;
   ALARM_SuppresionActiv := TRUE;
   ALARM_AlarmPresent := TRUE;
   StatusWork := 202;
   AlarmNo := 4;
   AlarmNo_Old := 4;
   OUT.AL_H := TRUE;
   OUT.WARN_L := TRUE;
   OUT.WARN_H := TRUE;
   MSW_EXT_AlarmFailUnAck := TRUE;
   MSW_Status_Trans := 202;
END_DATA_BLOCK

DATA_BLOCK "_2010CV180OA_DB"   // DB2218
TITLE = Instance DB Alarm: _100CV002S51
{ S7_Optimized_Access := 'FALSE' }
AUTHOR : METIS
NAME : ALARM_DB
VERSION : 8.0
// stored: InstanceOfName ACESYS_ALARM
"ACESYS_ALARM"
BEGIN
   FP_PARM.EnableTime_Low_Pre := 5;
   FP_EN.ParentSupress := TRUE;
   FP_EN.ParentSupressUnit := TRUE;
   SIG := FALSE;
   PWR := TRUE;
   EN_H := TRUE;
   OK := TRUE;
   AL_L := TRUE;
   AL_H := TRUE;
   WARN_L := TRUE;
   WARN_H := TRUE;
   MSW.EXT.Operation := TRUE;
   MSW.Status := 1;
   MSW.TimeStamp := 16#255D;
   BlockInfo.Ace_Version := 80;
   BlockInfo.Ace_BuildNo := 4;
   BlockInfo.State_Act := 1;
   BlockInfo.State_Prev := 202;
   BlockInfo.DB_Number := 2218;
   FP_PARM.EnableTime_Low_Acc := 5;
   FP_EN.Alarm_High := TRUE;
   FP_SIM.SIG_Enable := TRUE;
   FP_SIM.PWR_Enable := TRUE;
   ONS.SecPulse2 := TRUE;
   ONS.AL_L_Aux := TRUE;
   ONS.AL_H_Aux := TRUE;
   EnableTime_High_Done := TRUE;
   StatusWork := 1;
   EnableTime_Low_Mem := 5;
   OUT.OK := TRUE;
   OUT.AL_L := TRUE;
   OUT.AL_H := TRUE;
   OUT.WARN_L := TRUE;
   OUT.WARN_H := TRUE;
   MSW_Status_Trans := 1;
END_DATA_BLOCK

DATA_BLOCK "_2010CV300S01_DB"   // DB3000
TITLE = Instance DB Select: _2010CV300S01
{ S7_Optimized_Access := 'FALSE' }
AUTHOR : METIS
NAME : SEL_DB
VERSION : 8.0
// stored: InstanceOfName ACESYS_SELECT
"ACESYS_SELECT"
BEGIN
   SEL := TRUE;
   MSW.Status := 24578;
   BlockInfo.Ace_Version := 80;
   BlockInfo.Ace_BuildNo := 1;
   BlockInfo.DB_Number := 3000;
   FP_CMD.Select := TRUE;
   FP_DIM.Deselect := TRUE;
   Ons_Sel := TRUE;
   Ons_FP_Sel := TRUE;
   Ons_NegIncing := TRUE;
   StatusWork := 2;
   OUT.SEL := TRUE;
   MSW_Status_Trans := 24578;
END_DATA_BLOCK

DATA_BLOCK "_2010CV180S01_DB"   // DB3001
TITLE = Instance DB Select:
{ S7_Optimized_Access := 'FALSE' }
AUTHOR : METIS
NAME : SEL_DB
VERSION : 8.0
// stored: InstanceOfName ACESYS_SELECT
"ACESYS_SELECT"
BEGIN
   SEL := TRUE;
   MSW.Status := 24578;
   BlockInfo.Ace_Version := 80;
   BlockInfo.Ace_BuildNo := 1;
   BlockInfo.DB_Number := 3001;
   FP_CMD.Select := TRUE;
   FP_DIM.Deselect := TRUE;
   Ons_Sel := TRUE;
   Ons_FP_Sel := TRUE;
   Ons_NegIncing := TRUE;
   StatusWork := 2;
   OUT.SEL := TRUE;
   MSW_Status_Trans := 24578;
END_DATA_BLOCK

DATA_BLOCK "_2010OB190S01_DB"   // DB3002
TITLE = Instance DB Select:
{ S7_Optimized_Access := 'FALSE' }
AUTHOR : METIS
NAME : SEL_DB
VERSION : 8.0
// stored: InstanceOfName ACESYS_SELECT
"ACESYS_SELECT"
BEGIN
   SEL := TRUE;
   MSW.Status := 24578;
   BlockInfo.Ace_Version := 80;
   BlockInfo.Ace_BuildNo := 1;
   BlockInfo.DB_Number := 3002;
   FP_CMD.Select := TRUE;
   FP_DIM.Deselect := TRUE;
   Ons_Sel := TRUE;
   Ons_FP_Sel := TRUE;
   Ons_NegIncing := TRUE;
   StatusWork := 2;
   OUT.SEL := TRUE;
   MSW_Status_Trans := 24578;
END_DATA_BLOCK

DATA_BLOCK "_2010CV120S01_DB"   // DB3003
TITLE = Instance DB Select:
{ S7_Optimized_Access := 'FALSE' }
AUTHOR : METIS
NAME : SEL_DB
VERSION : 8.0
// stored: InstanceOfName ACESYS_SELECT
"ACESYS_SELECT"
BEGIN
   SEL := TRUE;
   MSW.Status := 24578;
   BlockInfo.Ace_Version := 80;
   BlockInfo.Ace_BuildNo := 1;
   BlockInfo.DB_Number := 3003;
   FP_CMD.Select := TRUE;
   FP_DIM.Deselect := TRUE;
   Ons_Sel := TRUE;
   Ons_FP_Sel := TRUE;
   Ons_NegIncing := TRUE;
   StatusWork := 2;
   OUT.SEL := TRUE;
   MSW_Status_Trans := 24578;
END_DATA_BLOCK

DATA_BLOCK "_2010CR150S01_DB"   // DB3004
TITLE = Instance DB Select:
{ S7_Optimized_Access := 'FALSE' }
AUTHOR : METIS
NAME : SEL_DB
VERSION : 8.0
// stored: InstanceOfName ACESYS_SELECT
"ACESYS_SELECT"
BEGIN
   SEL := TRUE;
   MSW.Status := 24578;
   BlockInfo.Ace_Version := 80;
   BlockInfo.Ace_BuildNo := 1;
   BlockInfo.DB_Number := 3004;
   FP_CMD.Select := TRUE;
   FP_DIM.Deselect := TRUE;
   Ons_Sel := TRUE;
   Ons_FP_Sel := TRUE;
   Ons_NegIncing := TRUE;
   StatusWork := 2;
   OUT.SEL := TRUE;
   MSW_Status_Trans := 24578;
END_DATA_BLOCK

DATA_BLOCK "_2010SC130S01_DB"   // DB3005
TITLE = Instance DB Select:
{ S7_Optimized_Access := 'FALSE' }
AUTHOR : METIS
NAME : SEL_DB
VERSION : 8.0
// stored: InstanceOfName ACESYS_SELECT
"ACESYS_SELECT"
BEGIN
   SEL := TRUE;
   MSW.Status := 24578;
   BlockInfo.Ace_Version := 80;
   BlockInfo.Ace_BuildNo := 1;
   BlockInfo.DB_Number := 3005;
   FP_CMD.Select := TRUE;
   FP_DIM.Deselect := TRUE;
   Ons_Sel := TRUE;
   Ons_FP_Sel := TRUE;
   Ons_NegIncing := TRUE;
   StatusWork := 2;
   OUT.SEL := TRUE;
   MSW_Status_Trans := 24578;
END_DATA_BLOCK

DATA_BLOCK "_2010BF110S01_DB"   // DB3006
TITLE = Instance DB Select: _2010BF110S01
{ S7_Optimized_Access := 'FALSE' }
AUTHOR : METIS
NAME : SEL_DB
VERSION : 8.0
// stored: InstanceOfName ACESYS_SELECT
"ACESYS_SELECT"
BEGIN
   SEL := TRUE;
   MSW.Status := 24578;
   BlockInfo.Ace_Version := 80;
   BlockInfo.Ace_BuildNo := 1;
   BlockInfo.DB_Number := 3006;
   FP_CMD.Select := TRUE;
   FP_DIM.Deselect := TRUE;
   Ons_Sel := TRUE;
   Ons_FP_Sel := TRUE;
   Ons_NegIncing := TRUE;
   StatusWork := 2;
   OUT.SEL := TRUE;
   MSW_Status_Trans := 24578;
END_DATA_BLOCK

DATA_BLOCK "_2090TK740Y01S01_DB"   // DB3007
{ S7_Optimized_Access := 'FALSE' }
AUTHOR : FLSmidth
FAMILY : ACESYS
NAME : SELECT
VERSION : 8.0
// stored: InstanceOfName ACESYS_SELECT
"ACESYS_SELECT"
BEGIN
END_DATA_BLOCK

DATA_BLOCK "_2090TK740Y03S01_DB"   // DB3008
{ S7_Optimized_Access := 'FALSE' }
AUTHOR : FLSmidth
FAMILY : ACESYS
NAME : SELECT
VERSION : 8.0
// stored: InstanceOfName ACESYS_SELECT
"ACESYS_SELECT"
BEGIN
END_DATA_BLOCK

DATA_BLOCK "_2090PU736U01S02_DB"   // DB3009
{ S7_Optimized_Access := 'FALSE' }
AUTHOR : FLSmidth
FAMILY : ACESYS
NAME : SELECT
VERSION : 8.0
// stored: InstanceOfName ACESYS_SELECT
"ACESYS_SELECT"
BEGIN
END_DATA_BLOCK

DATA_BLOCK "_2090TK649Y03S01_DB"   // DB3010
{ S7_Optimized_Access := 'FALSE' }
AUTHOR : FLSmidth
FAMILY : ACESYS
NAME : SELECT
VERSION : 8.0
// stored: InstanceOfName ACESYS_SELECT
"ACESYS_SELECT"
BEGIN
END_DATA_BLOCK

DATA_BLOCK "_2010SJ950M01S01_DB"   // DB3039
TITLE = Instance DB Select: _2010SJ950M01S01
{ S7_Optimized_Access := 'FALSE' }
AUTHOR : METIS
NAME : SEL_DB
VERSION : 8.0
// stored: InstanceOfName ACESYS_SELECT
"ACESYS_SELECT"
BEGIN
   FCOFF := TRUE;
   MSW.Status := 3;
   BlockInfo.Ace_Version := 80;
   BlockInfo.Ace_BuildNo := 1;
   BlockInfo.DB_Number := 3039;
   FP_CMD.DeSelect := TRUE;
   Ons_DeSel := TRUE;
   Ons_FP_DeSel := TRUE;
   Ons_NegIncing := TRUE;
   StatusWork := 3;
   MSW_Status_Trans := 3;
END_DATA_BLOCK

DATA_BLOCK "HLC_DB"   // DB4000
TITLE = Instance DB HLC: High-Level-Control
{ S7_Optimized_Access := 'FALSE' }
AUTHOR : METIS
FAMILY : ACESYS
NAME : HLCDB
VERSION : 8.0
// stored: InstanceOfName ACESYS_HLC
"ACESYS_HLC"
BEGIN
   DEPT_LINK.TimeStamp := 16#1261;
   DEPT_LINK.OB1_CycleTime := 62;
   DEPT_LINK.Pulse_1sec := TRUE;
   DEPT_LINK.Man_Enable := TRUE;
   DEPT_LINK.Loc_Enable := TRUE;
   DEPT_LINK.Test_Enable := TRUE;
   DEPT_LINK.SS_FP_Enable := TRUE;
   DEPT_LINK.EmergencyStop := TRUE;
   DEPT_LINK.All_Group_Sel_RDY := TRUE;
   DEPT_LINK.All_Selected_Running := TRUE;
   DEPT_LINK.Ready_For_StopCmd := TRUE;
   DEPT_LINK.SEC_Toggle := TRUE;
   CCA1 := FALSE;
   CCA2 := FALSE;
   GRP_01_RDY := FALSE;
   GRP_02_RDY := FALSE;
   GRP_03_RDY := FALSE;
   GRP_04_RDY := FALSE;
   GRP_05_RDY := FALSE;
   GRP_06_RDY := FALSE;
   GRP_07_RDY := FALSE;
   GRP_08_RDY := FALSE;
   GRP_09_RDY := FALSE;
   GRP_10_RDY := FALSE;
   MSW.EXT.AlarmPresent := TRUE;
   MSW.Status := 1;
   MSW.TimeStamp := 16#3928;
   BlockInfo.Ace_Version := 80;
   BlockInfo.Ace_BuildNo := 1;
   BlockInfo.DB_Number := 4000;
   FP_PARM.KA_Time_Actual := 60;
   ONS.OFF_01 := TRUE;
   ONS.OFF_02 := TRUE;
   ONS.OFF_03 := TRUE;
   ONS.OFF_04 := TRUE;
   ONS.OFF_05 := TRUE;
   ONS.OFF_06 := TRUE;
   ONS.OFF_07 := TRUE;
   ONS.OFF_08 := TRUE;
   ONS.OFF_09 := TRUE;
   ONS.OFF_10 := TRUE;
   ALARM_AlarmPresent := TRUE;
   StatusWork := 1;
   MSW_Status_Trans := 1;
END_DATA_BLOCK

DATA_BLOCK "_997CS100CPU_DB"   // DB4001
TITLE = Instance DB PLC Diag: PLC Diagnostic
{ S7_Optimized_Access := 'FALSE' }
AUTHOR : METIS
FAMILY : ACESYS
NAME : PLCDB
VERSION : 8.0
// stored: InstanceOfName ACESYS_PLC_DIAGV2
"ACESYS_PLC_DIAGV2"
BEGIN
   OB35_ScanTime_In := 100;
   CPU_Type := 400;
   Master_Link.Pulse_Sec := TRUE;
   Master_Link.SS_FP_Enable := TRUE;
   Master_Link.Man_Enable := TRUE;
   Master_Link.Loc_Enable := TRUE;
   Master_Link.Test_Enable := TRUE;
   Master_Link.SEC_Toggle := TRUE;
   Master_Link.TimeStamp := 16#B1BD;
   Master_Link.OB1_CycleTime := 61;
   Type_Fault := TRUE;
   CPUClock_Sec := 35;
   CPUClock_Min := 17;
   CPUClock_Hour := 5;
   CPUClock_Day := 22;
   CPUClock_Month := 6;
   CPUClock_Year := 24;
   OB01_ScanTime := 61;
   OB35_ScanTime := 100;
   Memory_Total := 264_184_832;
   Memory_Used := 11549696;
   Mem_UsePercentage := 4.371824;
   MSW.EXT.AlarmPresent := TRUE;
   MSW.EXT.AlarmFailUnAck := TRUE;
   MSW.Status := 112;
   MSW.TimeStamp := 16#228B;
   BlockInfo.Ace_Version := 80;
   BlockInfo.Ace_BuildNo := 1;
   BlockInfo.DB_Number := 4001;
   StatusWork := 112;
   Record_LED_MAINT := 16#0001;
   Record_LED_ERROR := 16#0004;
   AlarmNo := 2;
   AlarmNo_Old := 2;
   ALARM_AlarmPresent := TRUE;
   Spare25 := TRUE;
   CPU_RUN_IND := TRUE;
   OUT.Type_Fault := TRUE;
   MSW_Status_Trans := 112;
   GetSMCinfo_Instance.REQ := TRUE;
   GetSMCinfo_Instance.Done := TRUE;
   GetSMCinfo_Instance.Info := 257993;
   GetSMCinfo_Instance_1.REQ := TRUE;
   GetSMCinfo_Instance_1.Mode := 1;
   GetSMCinfo_Instance_1.Done := TRUE;
   GetSMCinfo_Instance_1.Info := 11279;
   GET_IM_DATA_Instance.LADDR := 50;
   GET_IM_DATA_Instance.ERROR := TRUE;
   GET_IM_DATA_Instance.STATUS := 16#8093;
   GET_IM_DATA_Instance.fbGETATTR.ID := 16#0000_0000;
   GET_IM_DATA_Instance.fbGETATTR.AID := 16#0000_0000;
   GET_IM_DATA_Instance.sdw_GetAttrID := 16#0000_0031;
   GET_IM_DATA_Instance.sdw_GetAttrAID := 16#0000_0EA9;
   GET_IM_DATA_Instance.sui_imdataLen_netto := 54;
   GET_IM_DATA_Instance.pa_DataChar[0] := ' ';
   GET_IM_DATA_Instance.pa_DataChar[1] := ' ';
   GET_IM_DATA_Instance.pa_DataChar[2] := ' ';
   GET_IM_DATA_Instance.pa_DataChar[3] := ' ';
   GET_IM_DATA_Instance.pa_DataChar[4] := ' ';
   GET_IM_DATA_Instance.pa_DataChar[5] := ' ';
   GET_IM_DATA_Instance.pa_DataChar[6] := ' ';
   GET_IM_DATA_Instance.pa_DataChar[7] := ' ';
   GET_IM_DATA_Instance.pa_DataChar[8] := ' ';
   GET_IM_DATA_Instance.pa_DataChar[9] := ' ';
   GET_IM_DATA_Instance.pa_DataChar[10] := ' ';
   GET_IM_DATA_Instance.pa_DataChar[11] := ' ';
   GET_IM_DATA_Instance.pa_DataChar[12] := ' ';
   GET_IM_DATA_Instance.pa_DataChar[13] := ' ';
   GET_IM_DATA_Instance.pa_DataChar[14] := ' ';
   GET_IM_DATA_Instance.pa_DataChar[15] := ' ';
   GET_IM_DATA_Instance.pa_DataChar[16] := ' ';
   GET_IM_DATA_Instance.pa_DataChar[17] := ' ';
   GET_IM_DATA_Instance.pa_DataChar[18] := ' ';
   GET_IM_DATA_Instance.pa_DataChar[19] := ' ';
   GET_IM_DATA_Instance.pa_DataChar[20] := ' ';
   GET_IM_DATA_Instance.pa_DataChar[21] := ' ';
   GET_IM_DATA_Instance.pa_DataChar[22] := ' ';
   GET_IM_DATA_Instance.pa_DataChar[23] := ' ';
   GET_IM_DATA_Instance.pa_DataChar[24] := ' ';
   GET_IM_DATA_Instance.pa_DataChar[25] := ' ';
   GET_IM_DATA_Instance.pa_DataChar[26] := ' ';
   GET_IM_DATA_Instance.pa_DataChar[27] := ' ';
   GET_IM_DATA_Instance.pa_DataChar[28] := ' ';
   GET_IM_DATA_Instance.pa_DataChar[29] := ' ';
   GET_IM_DATA_Instance.pa_DataChar[30] := ' ';
   GET_IM_DATA_Instance.pa_DataChar[31] := ' ';
   GET_IM_DATA_Instance.pa_DataChar[32] := ' ';
   GET_IM_DATA_Instance.pa_DataChar[33] := ' ';
   GET_IM_DATA_Instance.pa_DataChar[34] := ' ';
   GET_IM_DATA_Instance.pa_DataChar[35] := ' ';
   GET_IM_DATA_Instance.pa_DataChar[36] := ' ';
   GET_IM_DATA_Instance.pa_DataChar[37] := ' ';
   GET_IM_DATA_Instance.pa_DataChar[38] := ' ';
   GET_IM_DATA_Instance.pa_DataChar[39] := ' ';
   GET_IM_DATA_Instance.pa_DataChar[40] := ' ';
   GET_IM_DATA_Instance.pa_DataChar[41] := ' ';
   GET_IM_DATA_Instance.pa_DataChar[42] := ' ';
   GET_IM_DATA_Instance.pa_DataChar[43] := ' ';
   GET_IM_DATA_Instance.pa_DataChar[44] := ' ';
   GET_IM_DATA_Instance.pa_DataChar[45] := ' ';
   GET_IM_DATA_Instance.pa_DataChar[46] := ' ';
   GET_IM_DATA_Instance.pa_DataChar[47] := ' ';
   GET_IM_DATA_Instance.pa_DataChar[48] := ' ';
   GET_IM_DATA_Instance.pa_DataChar[49] := ' ';
   GET_IM_DATA_Instance.pa_DataChar[50] := ' ';
   GET_IM_DATA_Instance.pa_DataChar[51] := ' ';
   GET_IM_DATA_Instance.pa_DataChar[52] := ' ';
   GET_IM_DATA_Instance.pa_DataChar[53] := ' ';
   GET_IM_DATA_Instance.pa_TemporaryCharArray[0] := ' ';
   GET_IM_DATA_Instance.pa_TemporaryCharArray[1] := ' ';
   GET_IM_DATA_Instance.pa_TemporaryCharArray[2] := ' ';
   GET_IM_DATA_Instance.pa_TemporaryCharArray[3] := ' ';
   GET_IM_DATA_Instance.pa_TemporaryCharArray[4] := ' ';
   GET_IM_DATA_Instance.pa_TemporaryCharArray[5] := ' ';
   GET_IM_DATA_Instance.pa_TemporaryCharArray[6] := ' ';
   GET_IM_DATA_Instance.pa_TemporaryCharArray[7] := ' ';
   GET_IM_DATA_Instance.pa_TemporaryCharArray[8] := ' ';
   GET_IM_DATA_Instance.pa_TemporaryCharArray[9] := ' ';
   GET_IM_DATA_Instance.pa_TemporaryCharArray[10] := ' ';
   GET_IM_DATA_Instance.pa_TemporaryCharArray[11] := ' ';
   GET_IM_DATA_Instance.pa_TemporaryCharArray[12] := ' ';
   GET_IM_DATA_Instance.pa_TemporaryCharArray[13] := ' ';
   GET_IM_DATA_Instance.pa_TemporaryCharArray[14] := ' ';
   GET_IM_DATA_Instance.pa_TemporaryCharArray[15] := ' ';
   GET_IM_DATA_Instance.pa_TemporaryCharArray[16] := ' ';
   GET_IM_DATA_Instance.pa_TemporaryCharArray[17] := ' ';
   GET_IM_DATA_Instance.pa_TemporaryCharArray[18] := ' ';
   GET_IM_DATA_Instance.pa_TemporaryCharArray[19] := ' ';
END_DATA_BLOCK

DATA_BLOCK "_997CS100NETMCCVFD1_DB"   // DB4002
TITLE = Instance DB PLC Diag: PN Net Diagnostic MCCVFD1
{ S7_Optimized_Access := 'FALSE' }
AUTHOR : METIS
FAMILY : ACESYS
NAME : PNNET_DB
VERSION : 8.0
// stored: InstanceOfName ACESYS_PROFINET
"ACESYS_PROFINET"
BEGIN
   Master_Link.SS_FP_Enable := TRUE;
   Master_Link.Man_Enable := TRUE;
   Master_Link.Loc_Enable := TRUE;
   Master_Link.Test_Enable := TRUE;
   Master_Link.SEC_Toggle := TRUE;
   Master_Link.TimeStamp := 16#B1C2;
   Master_Link.OB1_CycleTime := 43;
   IO_System_CP := 105;
   MSW.EXT.AlarmPresent := TRUE;
   MSW.EXT.AlarmFailUnAck := TRUE;
   MSW.Status := 104;
   MSW.TimeStamp := 16#3928;
   BlockInfo.Ace_Version := 80;
   BlockInfo.Ace_BuildNo := 1;
   BlockInfo.DB_Number := 4002;
   READING_INDEX_FAILURE := TRUE;
   ALARM_AlarmPresent := TRUE;
   ConfigNodeAlarm := TRUE;
   AlarmNo := 4;
   AlarmNo_Old := 4;
   StatusWork := 104;
   MSW_Status_Trans := 104;
END_DATA_BLOCK

DATA_BLOCK "_997CS100NETPNIO_DB"   // DB4003
TITLE = Instance DB PLC Diag: PN Net Diagnostic PNIO
{ S7_Optimized_Access := 'FALSE' }
AUTHOR : METIS
FAMILY : ACESYS
NAME : PNNET_DB
VERSION : 8.0
// stored: InstanceOfName ACESYS_PROFINET
"ACESYS_PROFINET"
BEGIN
   Master_Link.SS_FP_Enable := TRUE;
   Master_Link.Man_Enable := TRUE;
   Master_Link.Loc_Enable := TRUE;
   Master_Link.Test_Enable := TRUE;
   Master_Link.SEC_Toggle := TRUE;
   Master_Link.TimeStamp := 16#B1C2;
   Master_Link.OB1_CycleTime := 43;
   IO_System_CP := 100;
   MSW.EXT.AlarmPresent := TRUE;
   MSW.EXT.AlarmFailUnAck := TRUE;
   MSW.Status := 105;
   MSW.TimeStamp := 16#3928;
   BlockInfo.Ace_Version := 80;
   BlockInfo.Ace_BuildNo := 1;
   BlockInfo.DB_Number := 4003;
   FP_PARM.SLAVES_AFFECTED_NUM := 12;
   FP_PARM.SLAVES_EXIST_NUM := 12;
   CONFIGURED[0] := TRUE;
   CONFIGURED[5] := TRUE;
   CONFIGURED[6] := TRUE;
   CONFIGURED[7] := TRUE;
   CONFIGURED[8] := TRUE;
   CONFIGURED[9] := TRUE;
   CONFIGURED[10] := TRUE;
   CONFIGURED[14] := TRUE;
   CONFIGURED[15] := TRUE;
   CONFIGURED[17] := TRUE;
   CONFIGURED[18] := TRUE;
   CONFIGURED[19] := TRUE;
   CONFIGURED[20] := TRUE;
   PRESENT[0] := TRUE;
   PRESENT[5] := TRUE;
   PRESENT[6] := TRUE;
   PRESENT[7] := TRUE;
   PRESENT[8] := TRUE;
   PRESENT[9] := TRUE;
   PRESENT[10] := TRUE;
   PRESENT[14] := TRUE;
   PRESENT[15] := TRUE;
   PRESENT[17] := TRUE;
   PRESENT[18] := TRUE;
   PRESENT[19] := TRUE;
   PRESENT[20] := TRUE;
   AFFECTED[0] := TRUE;
   AFFECTED[5] := TRUE;
   AFFECTED[6] := TRUE;
   AFFECTED[7] := TRUE;
   AFFECTED[8] := TRUE;
   AFFECTED[9] := TRUE;
   AFFECTED[10] := TRUE;
   AFFECTED[14] := TRUE;
   AFFECTED[15] := TRUE;
   AFFECTED[17] := TRUE;
   AFFECTED[18] := TRUE;
   AFFECTED[19] := TRUE;
   AFFECTED[20] := TRUE;
   READING_INDEX_FAILURE := TRUE;
   DR_Data[0] := 16#E1C7;
   DR_Data[1] := 16#1E00;
   ALARM_AlarmPresent := TRUE;
   NodeErrorAlarm := TRUE;
   AlarmNo := 5;
   AlarmNo_Old := 5;
   StatusWork := 105;
   MSW_Status_Trans := 105;
END_DATA_BLOCK

DATA_BLOCK "_997CS100NETSPLC_DB"   // DB4004
TITLE = Instance DB PLC Diag: PN Net Diagnostic SPLC
{ S7_Optimized_Access := 'FALSE' }
AUTHOR : METIS
FAMILY : ACESYS
NAME : PNNET_DB
VERSION : 8.0
// stored: InstanceOfName ACESYS_PROFINET
"ACESYS_PROFINET"
BEGIN
   Master_Link.SS_FP_Enable := TRUE;
   Master_Link.Man_Enable := TRUE;
   Master_Link.Loc_Enable := TRUE;
   Master_Link.Test_Enable := TRUE;
   Master_Link.SEC_Toggle := TRUE;
   Master_Link.TimeStamp := 16#B1C2;
   Master_Link.OB1_CycleTime := 43;
   IO_System_CP := 106;
   MSW.EXT.AlarmPresent := TRUE;
   MSW.EXT.AlarmFailUnAck := TRUE;
   MSW.Status := 104;
   MSW.TimeStamp := 16#3928;
   BlockInfo.Ace_Version := 80;
   BlockInfo.Ace_BuildNo := 1;
   BlockInfo.DB_Number := 4004;
   READING_INDEX_FAILURE := TRUE;
   ALARM_AlarmPresent := TRUE;
   ConfigNodeAlarm := TRUE;
   AlarmNo := 4;
   AlarmNo_Old := 4;
   StatusWork := 104;
   MSW_Status_Trans := 104;
END_DATA_BLOCK

DATA_BLOCK "_2010CV300U01_DB"   // DB4007
TITLE = Instance DB Unimotor: _2010CV300U01
{ S7_Optimized_Access := 'FALSE' }
AUTHOR : METIS
NAME : UNIMO_DB
VERSION : 8.0
// stored: InstanceOfName ACESYS_MOTOR
"ACESYS_MOTOR"
BEGIN
   FP_SEL.MD_OnOff := TRUE;
   FP_SEL.STW_Local := TRUE;
   FP_SEL.STW_Manual := TRUE;
   FP_SEL.STW_Single := TRUE;
   FP_SEL.Type_Unimotor := TRUE;
   FP_SEL.ParentCollection := TRUE;
   FP_EN.Mode_Auto := TRUE;
   FP_EN.Mode_Man := TRUE;
   FP_EN.PB_QStop := TRUE;
   FP_SHOW.AI1 := TRUE;
   FP_SHOW.OVL := TRUE;
   FP_SHOW.LSTP := TRUE;
   FP_SHOW.DRDY := TRUE;
   FP_SHOW.STALL := TRUE;
   FP_SHOW.EARTH := TRUE;
   FP_SHOW.UBAL := TRUE;
   FP_SHOW.GFA := TRUE;
   FP_SHOW.GWA := TRUE;
   FP_SHOW.BUSF := TRUE;
   FP_SHOW.DOPR := TRUE;
   FP_SHOW.DTEST := TRUE;
   FP_SHOW.ACK := TRUE;
   FP_SHOW.PB_Reset := TRUE;
   FP_PARM.StartWarn_Pre := 10;
   FP_PARM.RunDelay1_Pre := 5;
   FP_PARM.DelayStop_Pre := 60;
   FP_PARM.ReturnMon_Pre := 2;
   FP_PARM.SpeedMonOnDelay_Pre := 10;
   FP_PARM.SpeedMonOffDelay_Pre := 10;
   FP_PARM.LeaveFS_Pre := 5;
   FP_PARM.ReachLS_Pre := 30;
   FP_PARM.ReachFS_Pre := 10;
   FP_PARM.AI1_Max := 487.0;
   FP_PARM.AI2_Max := 100.0;
   FP_PARM.AI3_Max := 100.0;
   FP_PARM.AO1a_Max := 100.0;
   FP_PARM.AO2a_Max := 100.0;
   FP_PARM.AO3a_Max := 100.0;
   FP_PARM.AO1b_Max := 487.0;
   FP_PARM.AO2b_Max := 250.0;
   FP_PARM.AO3b_Max := 1489.0;
   CMD.GSEL := TRUE;
   RET1 := TRUE;
   SFS := FALSE;
   ES := TRUE;
   AI1 := 251.9;
   AI2 := 55.8;
   AI3 := 110.9;
   SPSET := 110.0;
   INTL.OK := TRUE;
   INTL.DetectFirst := TRUE;
   INTL.ClearFirst := TRUE;
   INTL_SEQ_STR1.OK := TRUE;
   INTL_SEQ_STR1.DetectFirst := TRUE;
   INTL_SEQ_STR1.ClearFirst := TRUE;
   INTL_SEQ_STR2.OK := TRUE;
   INTL_SEQ_STR2.ClearFirst := TRUE;
   INTL_SEQ_STP.OK := TRUE;
   CON1 := TRUE;
   LAMP1 := TRUE;
   SACK := TRUE;
   RD1 := TRUE;
   RUN1 := TRUE;
   OK := TRUE;
   AUT := TRUE;
   AO1a := 51.72484;
   AO1b := 251.9;
   AO2a := 55.8;
   AO2b := 139.5;
   AO3a := 110.9;
   AO3b := 1651.301;
   CV := 110.0;
   MSW.EXT.Operation := TRUE;
   MSW.Status := 4177;
   MSW.TimeStamp := 16#30DE;
   BlockInfo.Ace_Version := 80;
   BlockInfo.Ace_BuildNo := 13;
   BlockInfo.State_Act := 108;
   BlockInfo.State_Prev := 106;
   BlockInfo.DB_Number := 4007;
   FP_CMD.Auto := TRUE;
   FP_SEL.MD := TRUE;
   FP_DIM.Reset := TRUE;
   FP_SHOW.PB_Auto := TRUE;
   FP_SHOW.PB_Manual := TRUE;
   FP_SHOW.PB_Start1 := TRUE;
   FP_SHOW.PB_Stop := TRUE;
   FP_SHOW.AI2 := TRUE;
   FP_SHOW.AI3 := TRUE;
   FP_SHOW.SP := TRUE;
   FP_SHOW.MCC := TRUE;
   FP_SHOW.RDY := TRUE;
   FP_SHOW.SSW := TRUE;
   FP_SHOW.ES := TRUE;
   FP_SHOW.TFA := TRUE;
   FP_SHOW.MD := TRUE;
   FP_SHOW.ASTR := TRUE;
   FP_PARM.StartWarn_Acc := 10;
   FP_PARM.RunDelay1_Acc := 5;
   FP_PARM.DelayStop_Acc := 60;
   FP_PARM.ReturnMon_Acc := 2;
   FP_PARM.SpeedMonOnDelay_Acc := 10;
   FP_PARM.SpeedMonOffDelay_Acc := 10;
   FP_PARM.LeaveFS_Acc := 5;
   FP_PARM.ReachLS_Acc := 30;
   FP_PARM.ReachFS_Acc := 10;
   FP_PARM.MD_Freq_SP := 1;
   FP_PARM.INTL := TRUE;
   FP_PARM.INTL_SEQ_STR1 := TRUE;
   FP_PARM.INTL_SEQ_STR2 := TRUE;
   FP_SIM.OVL_Enable := TRUE;
   FP_SIM.RDY_Enable := TRUE;
   FP_SIM.SSW_Enable := TRUE;
   FP_SIM.TFA_Enable := TRUE;
   FP_SIM.MCC_Enable := TRUE;
   FP_SIM.DRDY_Enable := TRUE;
   FP_SIM.MD_Enable := TRUE;
   FP_SIM.GFA_Enable := TRUE;
   FP_SIM.GWA_Enable := TRUE;
   FP_SIM.STALL_Enable := TRUE;
   FP_SIM.EARTH_Enable := TRUE;
   FP_SIM.UBAL_Enable := TRUE;
   FP_SIM.BUSF_Enable := TRUE;
   FP_SIM.RET1_Enable := TRUE;
   FP_SIM.RET2_Enable := TRUE;
   FP_SIM.DOPR_Enable := TRUE;
   FP_SIM.ACK_Enable := TRUE;
   FP_SIM.LSTP_Enable := TRUE;
   FP_SIM.REM_Enable := TRUE;
   FP_SIM.SFS_Enable := TRUE;
   FP_SIM.SLS_Enable := TRUE;
   FP_SIM.ES_Enable := TRUE;
   FP_SIM.WORK.Flash_Slow := TRUE;
   FP_SIM.WORK.CON1 := TRUE;
   AdapterBlock.Intell_Type := 282;
   AdapterBlock.VersionNo := 220;
   AdapterBlock.FuncType := 41;
   AdapterBlock.NetNo := 101;
   AdapterBlock.NodeNo := 3;
   AdapterBlock.Flash_Slow := TRUE;
   AdapterBlock.CON1 := TRUE;
   AdapterBlock.HMI_INT[1] := 5545;
   AdapterBlock.HMI_INT[6] := -395;
   AdapterBlock.HMI_INT[7] := 5500;
   AdapterBlock.HMI_INT[9] := 2;
   AdapterBlock.HMI_INT[10] := 2;
   AdapterBlock.HMI_INT[11] := 1;
   AdapterBlock.HMI_REAL[1] := 110.9;
   AdapterBlock.HMI_REAL[2] := 55.9;
   AdapterBlock.HMI_REAL[3] := 55.9;
   AdapterBlock.HMI_REAL[4] := 252.8;
   AdapterBlock.HMI_REAL[9] := 100.0;
   AdapterBlock.HMI_REAL[10] := 100.0;
   AdapterBlock.HMI_REAL[11] := 559.0;
   AdapterBlock.HMI_REAL[12] := 100.0;
   AdapterBlock.HMI_REAL[13] := 2528.0;
   AdapterBlock.HMI_BOOL[2] := TRUE;
   AdapterBlock.HMI_BOOL[9] := TRUE;
   AdapterBlock.HMI_BOOL[15] := TRUE;
   AdapterBlock.HMI_BOOL[33] := TRUE;
   AdapterBlock.HMI_BOOL[89] := TRUE;
   STATE.A_Running1 := TRUE;
   ONS.Unimotor := TRUE;
   ONS.MD_OnOff := TRUE;
   ONS.Cmd_Auto := TRUE;
   ONS.GLTP := TRUE;
   ONS.RET1 := TRUE;
   ONS.MD_Pulse := TRUE;
   ONS.CMD_Start1 := TRUE;
   ONS.CMD_Start2 := TRUE;
   ONS.SecPulse1 := TRUE;
   StatusWork := 81;
   ModePointer := 51;
   StartWarn_Mem := 10;
   DelayStop_Mem := 60;
   ReturnMon_Mem := 2;
   SpeedMonOffDelay_Mem := 10;
   LeaveFS_Mem := 5;
   ReachLS_Mem := 30;
   ReachFS_Mem := 10;
   ModeAuto := TRUE;
   Select := TRUE;
   FromStateAuto := TRUE;
   Rundelay1_Done := TRUE;
   SpeedMonOnDelay_Done := TRUE;
   ChangeDir2_Done := TRUE;
   RET1_OneScan := TRUE;
   OUT.CON1 := TRUE;
   OUT.LAMP1 := TRUE;
   OUT.SACK := TRUE;
   OUT.RD1 := TRUE;
   OUT.RUN1 := TRUE;
   OUT.OK := TRUE;
   OUT.AUT := TRUE;
   OUT.INTL_OK_STAT := TRUE;
   OUT.INTL_SEQ_STR1_OK_STAT := TRUE;
   OUT.INTL_SEQ_STR2_OK_STAT := TRUE;
   MSW_Status_Trans := 4177;
END_DATA_BLOCK

DATA_BLOCK "_2010CV180U01_DB"   // DB4008
TITLE = Instance DB Unimotor: _2010CV180U0
{ S7_Optimized_Access := 'FALSE' }
AUTHOR : METIS
NAME : UNIMO_DB
VERSION : 8.0
// stored: InstanceOfName ACESYS_MOTOR
"ACESYS_MOTOR"
BEGIN
   FP_SEL.STW_Local := TRUE;
   FP_SEL.STW_Manual := TRUE;
   FP_SEL.STW_Single := TRUE;
   FP_SEL.Type_Unimotor := TRUE;
   FP_SEL.ParentCollection := TRUE;
   FP_EN.Mode_Auto := TRUE;
   FP_EN.Mode_Man := TRUE;
   FP_EN.PB_QStop := TRUE;
   FP_SHOW.AI1 := TRUE;
   FP_SHOW.OVL := TRUE;
   FP_SHOW.LSTP := TRUE;
   FP_SHOW.DRDY := TRUE;
   FP_SHOW.STALL := TRUE;
   FP_SHOW.EARTH := TRUE;
   FP_SHOW.UBAL := TRUE;
   FP_SHOW.GFA := TRUE;
   FP_SHOW.GWA := TRUE;
   FP_SHOW.BUSF := TRUE;
   FP_SHOW.DOPR := TRUE;
   FP_SHOW.DTEST := TRUE;
   FP_SHOW.ACK := TRUE;
   FP_SHOW.PB_Reset := TRUE;
   FP_PARM.StartWarn_Pre := 15;
   FP_PARM.RunDelay1_Pre := 5;
   FP_PARM.DelayStop_Pre := 60;
   FP_PARM.ReturnMon_Pre := 2;
   FP_PARM.SpeedMonOnDelay_Pre := 10;
   FP_PARM.SpeedMonOffDelay_Pre := 10;
   FP_PARM.LeaveFS_Pre := 5;
   FP_PARM.ReachLS_Pre := 30;
   FP_PARM.ReachFS_Pre := 10;
   FP_PARM.AI1_Max := 58.7;
   FP_PARM.AI2_Max := 100.0;
   FP_PARM.AI3_Max := 100.0;
   FP_PARM.AO1a_Max := 100.0;
   FP_PARM.AO2a_Max := 100.0;
   FP_PARM.AO3a_Max := 100.0;
   FP_PARM.AO1b_Max := 58.7;
   FP_PARM.AO2b_Max := 30.0;
   FP_PARM.AO3b_Max := 1477.0;
   CMD.GSEL := TRUE;
   RET1 := TRUE;
   MD := FALSE;
   SFS := FALSE;
   ES := TRUE;
   AI1 := 63.6;
   AI2 := 30.6;
   AI3 := 90.0;
   SPSET := 90.0;
   INTL.OK := TRUE;
   INTL.DetectFirst := TRUE;
   INTL.ClearFirst := TRUE;
   INTL_SEQ_STR1.OK := TRUE;
   INTL_SEQ_STR1.DetectFirst := TRUE;
   INTL_SEQ_STR1.ClearFirst := TRUE;
   INTL_SEQ_STR2.OK := TRUE;
   INTL_SEQ_STR2.ClearFirst := TRUE;
   INTL_SEQ_STP.OK := TRUE;
   CON1 := TRUE;
   LAMP1 := TRUE;
   SACK := TRUE;
   RD1 := TRUE;
   RUN1 := TRUE;
   OK := TRUE;
   AUT := TRUE;
   AO1a := 108.3475;
   AO1b := 63.6;
   AO2a := 30.6;
   AO2b := 9.18;
   AO3a := 90.0;
   AO3b := 1329.3;
   CV := 90.0;
   MSW.EXT.Operation := TRUE;
   MSW.Status := 4177;
   MSW.TimeStamp := 16#3337;
   BlockInfo.Ace_Version := 80;
   BlockInfo.Ace_BuildNo := 13;
   BlockInfo.State_Act := 108;
   BlockInfo.State_Prev := 106;
   BlockInfo.DB_Number := 4008;
   FP_CMD.Auto := TRUE;
   FP_SEL.MD := TRUE;
   FP_SEL.MD_Puls := TRUE;
   FP_DIM.Reset := TRUE;
   FP_SHOW.PB_Auto := TRUE;
   FP_SHOW.PB_Manual := TRUE;
   FP_SHOW.PB_Start1 := TRUE;
   FP_SHOW.PB_Stop := TRUE;
   FP_SHOW.AI2 := TRUE;
   FP_SHOW.AI3 := TRUE;
   FP_SHOW.SP := TRUE;
   FP_SHOW.MCC := TRUE;
   FP_SHOW.RDY := TRUE;
   FP_SHOW.REM := TRUE;
   FP_SHOW.SSW := TRUE;
   FP_SHOW.ES := TRUE;
   FP_SHOW.TFA := TRUE;
   FP_SHOW.MD := TRUE;
   FP_SHOW.ASTR := TRUE;
   FP_PARM.StartWarn_Acc := 15;
   FP_PARM.RunDelay1_Acc := 5;
   FP_PARM.DelayStop_Acc := 60;
   FP_PARM.ReturnMon_Acc := 2;
   FP_PARM.SpeedMonOnDelay_Acc := 10;
   FP_PARM.SpeedMonOffDelay_Acc := 10;
   FP_PARM.SpeedMonTrigDelay_Pre := 10;
   FP_PARM.SpeedMonTrigDelay_Acc := 10;
   FP_PARM.LeaveFS_Acc := 5;
   FP_PARM.ReachLS_Acc := 30;
   FP_PARM.ReachFS_Acc := 10;
   FP_PARM.MD_Freq_SP := 30;
   FP_PARM.MD_Freq_PV := 209;
   FP_PARM.INTL := TRUE;
   FP_PARM.INTL_SEQ_STR1 := TRUE;
   FP_PARM.INTL_SEQ_STR2 := TRUE;
   FP_SIM.OVL_Enable := TRUE;
   FP_SIM.RDY_Enable := TRUE;
   FP_SIM.SSW_Enable := TRUE;
   FP_SIM.TFA_Enable := TRUE;
   FP_SIM.MCC_Enable := TRUE;
   FP_SIM.DRDY_Enable := TRUE;
   FP_SIM.MD_Enable := TRUE;
   FP_SIM.GFA_Enable := TRUE;
   FP_SIM.GWA_Enable := TRUE;
   FP_SIM.STALL_Enable := TRUE;
   FP_SIM.EARTH_Enable := TRUE;
   FP_SIM.UBAL_Enable := TRUE;
   FP_SIM.BUSF_Enable := TRUE;
   FP_SIM.RET1_Enable := TRUE;
   FP_SIM.RET2_Enable := TRUE;
   FP_SIM.DOPR_Enable := TRUE;
   FP_SIM.ACK_Enable := TRUE;
   FP_SIM.LSTP_Enable := TRUE;
   FP_SIM.REM_Enable := TRUE;
   FP_SIM.SFS_Enable := TRUE;
   FP_SIM.SLS_Enable := TRUE;
   FP_SIM.ES_Enable := TRUE;
   FP_SIM.WORK.Flash_Slow := TRUE;
   FP_SIM.WORK.CON1 := TRUE;
   FP_SIM.WORK.MD_Type_Puls := TRUE;
   AdapterBlock.Intell_Type := 282;
   AdapterBlock.VersionNo := 220;
   AdapterBlock.FuncType := 41;
   AdapterBlock.NetNo := 101;
   AdapterBlock.NodeNo := 3;
   AdapterBlock.Flash_Slow := TRUE;
   AdapterBlock.CON1 := TRUE;
   AdapterBlock.HMI_INT[1] := 4500;
   AdapterBlock.HMI_INT[6] := -312;
   AdapterBlock.HMI_INT[7] := 4500;
   AdapterBlock.HMI_INT[9] := 2;
   AdapterBlock.HMI_INT[10] := 2;
   AdapterBlock.HMI_INT[11] := 1;
   AdapterBlock.HMI_REAL[1] := 90.0;
   AdapterBlock.HMI_REAL[2] := 30.5;
   AdapterBlock.HMI_REAL[3] := 30.5;
   AdapterBlock.HMI_REAL[4] := 63.6;
   AdapterBlock.HMI_REAL[9] := 100.0;
   AdapterBlock.HMI_REAL[10] := 100.0;
   AdapterBlock.HMI_REAL[11] := 305.0;
   AdapterBlock.HMI_REAL[12] := 100.0;
   AdapterBlock.HMI_REAL[13] := 636.0;
   AdapterBlock.HMI_BOOL[2] := TRUE;
   AdapterBlock.HMI_BOOL[9] := TRUE;
   AdapterBlock.HMI_BOOL[15] := TRUE;
   AdapterBlock.HMI_BOOL[33] := TRUE;
   AdapterBlock.HMI_BOOL[89] := TRUE;
   STATE.A_Running1 := TRUE;
   ONS.Unimotor := TRUE;
   ONS.MD_Puls := TRUE;
   ONS.Cmd_Auto := TRUE;
   ONS.GLTP := TRUE;
   ONS.RET1 := TRUE;
   ONS.CMD_Start1 := TRUE;
   ONS.CMD_Start2 := TRUE;
   ONS.SecPulse1 := TRUE;
   StatusWork := 81;
   ModePointer := 51;
   StartWarn_Mem := 15;
   DelayStop_Mem := 60;
   ReturnMon_Mem := 2;
   SpeedMonOffDelay_Mem := 10;
   SpeedMonTrigDelay_Mem := 10;
   LeaveFS_Mem := 5;
   ReachLS_Mem := 30;
   ReachFS_Mem := 10;
   MD_Time := 287;
   MD_Time_DINT := 122;
   MD_Timer.ST := T#13D_5H_9M_951MS;
   MD_Timer.PT := T#10M;
   MD_Timer.RU := TRUE;
   MD_Timer.IN := TRUE;
   ModeAuto := TRUE;
   Select := TRUE;
   FromStateAuto := TRUE;
   Rundelay1_Done := TRUE;
   SpeedMonOnDelay_Done := TRUE;
   ChangeDir2_Done := TRUE;
   RET1_OneScan := TRUE;
   OUT.CON1 := TRUE;
   OUT.LAMP1 := TRUE;
   OUT.SACK := TRUE;
   OUT.RD1 := TRUE;
   OUT.RUN1 := TRUE;
   OUT.OK := TRUE;
   OUT.AUT := TRUE;
   OUT.INTL_OK_STAT := TRUE;
   OUT.INTL_SEQ_STR1_OK_STAT := TRUE;
   OUT.INTL_SEQ_STR2_OK_STAT := TRUE;
   MSW_Status_Trans := 4177;
END_DATA_BLOCK

DATA_BLOCK "_2010CV120M01_DB"   // DB4009
TITLE = Instance DB Unimotor: _2010CV120M01
{ S7_Optimized_Access := 'FALSE' }
AUTHOR : 7Art
NAME : UNIMO_DB
VERSION : 8.0
// stored: InstanceOfName ACESYS_MOTOR
"ACESYS_MOTOR"
BEGIN
   FP_SEL.MD_OnOff := TRUE;
   FP_SEL.STW_Local := TRUE;
   FP_SEL.STW_Manual := TRUE;
   FP_SEL.STW_Single := TRUE;
   FP_SEL.Type_Unimotor := TRUE;
   FP_SEL.ParentCollection := TRUE;
   FP_EN.Mode_Auto := TRUE;
   FP_EN.Mode_Man := TRUE;
   FP_EN.PB_QStop := TRUE;
   FP_SHOW.AI1 := TRUE;
   FP_SHOW.OVL := TRUE;
   FP_SHOW.DRDY := TRUE;
   FP_SHOW.STALL := TRUE;
   FP_SHOW.EARTH := TRUE;
   FP_SHOW.UBAL := TRUE;
   FP_SHOW.GFA := TRUE;
   FP_SHOW.GWA := TRUE;
   FP_SHOW.BUSF := TRUE;
   FP_SHOW.DOPR := TRUE;
   FP_SHOW.DTEST := TRUE;
   FP_SHOW.ACK := TRUE;
   FP_SHOW.PB_Reset := TRUE;
   FP_PARM.StartWarn_Pre := 15;
   FP_PARM.RunDelay1_Pre := 5;
   FP_PARM.DelayStop_Pre := 15;
   FP_PARM.ReturnMon_Pre := 2;
   FP_PARM.SpeedMonOnDelay_Pre := 10;
   FP_PARM.SpeedMonOffDelay_Pre := 10;
   FP_PARM.LeaveFS_Pre := 5;
   FP_PARM.ReachLS_Pre := 30;
   FP_PARM.ReachFS_Pre := 10;
   FP_PARM.AI1_Max := 100.0;
   FP_PARM.AI2_Max := 100.0;
   FP_PARM.AI3_Max := 100.0;
   FP_PARM.AO1a_Max := 100.0;
   FP_PARM.AO2a_Max := 100.0;
   FP_PARM.AO3a_Max := 100.0;
   FP_PARM.AO1b_Max := 14.0;
   FP_PARM.AO2b_Max := 100.0;
   FP_PARM.AO3b_Max := 100.0;
   CMD.GSEL := TRUE;
   RET1 := TRUE;
   MD := FALSE;
   SFS := FALSE;
   ES := TRUE;
   AI1 := 25.0;
   INTL.OK := TRUE;
   INTL.DetectFirst := TRUE;
   INTL.ClearFirst := TRUE;
   INTL_SEQ_STR1.OK := TRUE;
   INTL_SEQ_STR1.DetectFirst := TRUE;
   INTL_SEQ_STR1.ClearFirst := TRUE;
   INTL_SEQ_STR2.OK := TRUE;
   INTL_SEQ_STR2.ClearFirst := TRUE;
   INTL_SEQ_STP.OK := TRUE;
   CON1 := TRUE;
   LAMP1 := TRUE;
   SACK := TRUE;
   RD1 := TRUE;
   RUN1 := TRUE;
   OK := TRUE;
   AUT := TRUE;
   AO1a := 25.0;
   AO1b := 3.5;
   MSW.EXT.Operation := TRUE;
   MSW.Status := 4177;
   MSW.TimeStamp := 16#36C9;
   BlockInfo.Ace_Version := 80;
   BlockInfo.Ace_BuildNo := 13;
   BlockInfo.State_Act := 108;
   BlockInfo.State_Prev := 106;
   BlockInfo.DB_Number := 4009;
   FP_CMD.Auto := TRUE;
   FP_DIM.Reset := TRUE;
   FP_SHOW.PB_Auto := TRUE;
   FP_SHOW.PB_Manual := TRUE;
   FP_SHOW.PB_Start1 := TRUE;
   FP_SHOW.PB_Stop := TRUE;
   FP_PARM.StartWarn_Acc := 15;
   FP_PARM.RunDelay1_Acc := 5;
   FP_PARM.DelayStart_Pre := 5;
   FP_PARM.DelayStart_Acc := 5;
   FP_PARM.DelayStop_Acc := 15;
   FP_PARM.ReturnMon_Acc := 2;
   FP_PARM.SpeedMonOnDelay_Acc := 10;
   FP_PARM.SpeedMonOffDelay_Acc := 10;
   FP_PARM.LeaveFS_Acc := 5;
   FP_PARM.ReachLS_Acc := 30;
   FP_PARM.ReachFS_Acc := 10;
   FP_PARM.MD_Freq_SP := 1;
   FP_PARM.INTL := TRUE;
   FP_PARM.INTL_SEQ_STR1 := TRUE;
   FP_PARM.INTL_SEQ_STR2 := TRUE;
   FP_SIM.OVL_Enable := TRUE;
   FP_SIM.RDY_Enable := TRUE;
   FP_SIM.SSW_Enable := TRUE;
   FP_SIM.TFA_Enable := TRUE;
   FP_SIM.MCC_Enable := TRUE;
   FP_SIM.DRDY_Enable := TRUE;
   FP_SIM.MD_Enable := TRUE;
   FP_SIM.GFA_Enable := TRUE;
   FP_SIM.GWA_Enable := TRUE;
   FP_SIM.STALL_Enable := TRUE;
   FP_SIM.EARTH_Enable := TRUE;
   FP_SIM.UBAL_Enable := TRUE;
   FP_SIM.BUSF_Enable := TRUE;
   FP_SIM.RET1_Enable := TRUE;
   FP_SIM.RET2_Enable := TRUE;
   FP_SIM.DOPR_Enable := TRUE;
   FP_SIM.ACK_Enable := TRUE;
   FP_SIM.LSTP_Enable := TRUE;
   FP_SIM.REM_Enable := TRUE;
   FP_SIM.SFS_Enable := TRUE;
   FP_SIM.SLS_Enable := TRUE;
   FP_SIM.ES_Enable := TRUE;
   FP_SIM.WORK.Flash_Slow := TRUE;
   FP_SIM.WORK.CON1 := TRUE;
   AdapterBlock.Intell_Type := 54;
   AdapterBlock.VersionNo := 420;
   AdapterBlock.BuildNo := 1;
   AdapterBlock.FuncType := 41;
   AdapterBlock.NetNo := 101;
   AdapterBlock.NodeNo := 25;
   AdapterBlock.Flash_Slow := TRUE;
   AdapterBlock.CON1 := TRUE;
   AdapterBlock.HMI_INT[3] := 3;
   AdapterBlock.HMI_INT[5] := 2527;
   AdapterBlock.HMI_INT[6] := 474;
   AdapterBlock.HMI_INT[7] := 3000;
   AdapterBlock.HMI_INT[9] := 7168;
   AdapterBlock.HMI_INT[17] := 32020;
   AdapterBlock.HMI_INT[26] := 25;
   AdapterBlock.HMI_REAL[2] := 1400.0;
   AdapterBlock.HMI_BOOL[1] := TRUE;
   AdapterBlock.HMI_BOOL[4] := TRUE;
   AdapterBlock.HMI_BOOL[8] := TRUE;
   AdapterBlock.HMI_BOOL[17] := TRUE;
   AdapterBlock.HMI_BOOL[19] := TRUE;
   AdapterBlock.HMI_BOOL[20] := TRUE;
   AdapterBlock.HMI_BOOL[21] := TRUE;
   AdapterBlock.HMI_BOOL[28] := TRUE;
   AdapterBlock.HMI_BOOL[58] := TRUE;
   AdapterBlock.HMI_BOOL[66] := TRUE;
   AdapterBlock.HMI_BOOL[73] := TRUE;
   AdapterBlock.HMI_BOOL[77] := TRUE;
   AdapterBlock.HMI_BOOL[79] := TRUE;
   AdapterBlock.HMI_BOOL[92] := TRUE;
   AdapterBlock.HMI_BOOL[93] := TRUE;
   AdapterBlock.HMI_BOOL[98] := TRUE;
   AdapterBlock.HMI_BOOL[106] := TRUE;
   STATE.A_Running1 := TRUE;
   ONS.Unimotor := TRUE;
   ONS.MD_OnOff := TRUE;
   ONS.Cmd_Auto := TRUE;
   ONS.GLTP := TRUE;
   ONS.RET1 := TRUE;
   ONS.CMD_Start1 := TRUE;
   ONS.CMD_Start2 := TRUE;
   ONS.SecPulse1 := TRUE;
   StatusWork := 81;
   ModePointer := 51;
   StartWarn_Mem := 15;
   DelayStart_Mem := 5;
   DelayStop_Mem := 15;
   ReturnMon_Mem := 2;
   SpeedMonOnDelay_Mem := 10;
   SpeedMonOffDelay_Mem := 10;
   LeaveFS_Mem := 5;
   ReachLS_Mem := 30;
   ReachFS_Mem := 10;
   ModeAuto := TRUE;
   Select := TRUE;
   FromStateAuto := TRUE;
   Rundelay1_Done := TRUE;
   ChangeDir2_Done := TRUE;
   RET1_OneScan := TRUE;
   OUT.CON1 := TRUE;
   OUT.LAMP1 := TRUE;
   OUT.SACK := TRUE;
   OUT.RD1 := TRUE;
   OUT.RUN1 := TRUE;
   OUT.OK := TRUE;
   OUT.AUT := TRUE;
   OUT.INTL_OK_STAT := TRUE;
   OUT.INTL_SEQ_STR1_OK_STAT := TRUE;
   OUT.INTL_SEQ_STR2_OK_STAT := TRUE;
   MSW_Status_Trans := 4177;
END_DATA_BLOCK

DATA_BLOCK "_2010OB190M01_DB"   // DB4010
TITLE = Instance DB Unimotor: _2010CV180U0
{ S7_Optimized_Access := 'FALSE' }
AUTHOR : METIS
NAME : UNIMO_DB
VERSION : 8.0
// stored: InstanceOfName ACESYS_MOTOR
"ACESYS_MOTOR"
BEGIN
   FP_SEL.MD_OnOff := TRUE;
   FP_SEL.STW_Local := TRUE;
   FP_SEL.STW_Manual := TRUE;
   FP_SEL.STW_Single := TRUE;
   FP_SEL.Type_Unimotor := TRUE;
   FP_SEL.ParentCollection := TRUE;
   FP_EN.Mode_Auto := TRUE;
   FP_EN.Mode_Man := TRUE;
   FP_EN.PB_QStop := TRUE;
   FP_SHOW.PB_Reset := TRUE;
   FP_PARM.StartWarn_Pre := 15;
   FP_PARM.RunDelay1_Pre := 5;
   FP_PARM.DelayStop_Pre := 5;
   FP_PARM.ReturnMon_Pre := 2;
   FP_PARM.SpeedMonOnDelay_Pre := 10;
   FP_PARM.SpeedMonOffDelay_Pre := 10;
   FP_PARM.LeaveFS_Pre := 5;
   FP_PARM.ReachLS_Pre := 30;
   FP_PARM.ReachFS_Pre := 10;
   FP_PARM.AI1_Max := 100.0;
   FP_PARM.AI2_Max := 100.0;
   FP_PARM.AI3_Max := 100.0;
   FP_PARM.AO1a_Max := 100.0;
   FP_PARM.AO2a_Max := 100.0;
   FP_PARM.AO3a_Max := 100.0;
   FP_PARM.AO1b_Max := 100.0;
   FP_PARM.AO2b_Max := 100.0;
   FP_PARM.AO3b_Max := 100.0;
   CMD.GSEL := TRUE;
   RET1 := TRUE;
   SFS := FALSE;
   ES := TRUE;
   INTL.OK := TRUE;
   INTL.DetectFirst := TRUE;
   INTL.ClearFirst := TRUE;
   INTL_SEQ_STR1.OK := TRUE;
   INTL_SEQ_STR1.DetectFirst := TRUE;
   INTL_SEQ_STR1.ClearFirst := TRUE;
   INTL_SEQ_STR2.OK := TRUE;
   INTL_SEQ_STR2.ClearFirst := TRUE;
   INTL_SEQ_STP.OK := TRUE;
   CON1 := TRUE;
   LAMP1 := TRUE;
   SACK := TRUE;
   RD1 := TRUE;
   RUN1 := TRUE;
   OK := TRUE;
   AUT := TRUE;
   RES := TRUE;
   MSW.EXT.Operation := TRUE;
   MSW.Status := 4177;
   MSW.TimeStamp := 16#32DC;
   BlockInfo.Ace_Version := 80;
   BlockInfo.Ace_BuildNo := 13;
   BlockInfo.State_Act := 108;
   BlockInfo.State_Prev := 106;
   BlockInfo.DB_Number := 4010;
   FP_CMD.Auto := TRUE;
   FP_DIM.Reset := TRUE;
   FP_SHOW.PB_Auto := TRUE;
   FP_SHOW.PB_Manual := TRUE;
   FP_SHOW.PB_Start1 := TRUE;
   FP_SHOW.PB_Stop := TRUE;
   FP_SHOW.MCC := TRUE;
   FP_PARM.StartWarn_Acc := 15;
   FP_PARM.RunDelay1_Acc := 5;
   FP_PARM.DelayStop_Acc := 5;
   FP_PARM.ReturnMon_Acc := 2;
   FP_PARM.SpeedMonOnDelay_Acc := 10;
   FP_PARM.SpeedMonOffDelay_Acc := 10;
   FP_PARM.LeaveFS_Acc := 5;
   FP_PARM.ReachLS_Acc := 30;
   FP_PARM.ReachFS_Acc := 10;
   FP_PARM.MD_Freq_SP := 1;
   FP_PARM.INTL := TRUE;
   FP_PARM.INTL_SEQ_STR1 := TRUE;
   FP_PARM.INTL_SEQ_STR2 := TRUE;
   FP_SIM.OVL_Enable := TRUE;
   FP_SIM.RDY_Enable := TRUE;
   FP_SIM.SSW_Enable := TRUE;
   FP_SIM.TFA_Enable := TRUE;
   FP_SIM.MCC_Enable := TRUE;
   FP_SIM.DRDY_Enable := TRUE;
   FP_SIM.MD_Enable := TRUE;
   FP_SIM.GFA_Enable := TRUE;
   FP_SIM.GWA_Enable := TRUE;
   FP_SIM.STALL_Enable := TRUE;
   FP_SIM.EARTH_Enable := TRUE;
   FP_SIM.UBAL_Enable := TRUE;
   FP_SIM.BUSF_Enable := TRUE;
   FP_SIM.RET1_Enable := TRUE;
   FP_SIM.RET2_Enable := TRUE;
   FP_SIM.DOPR_Enable := TRUE;
   FP_SIM.ACK_Enable := TRUE;
   FP_SIM.LSTP_Enable := TRUE;
   FP_SIM.REM_Enable := TRUE;
   FP_SIM.SFS_Enable := TRUE;
   FP_SIM.SLS_Enable := TRUE;
   FP_SIM.ES_Enable := TRUE;
   FP_SIM.WORK.Flash_Slow := TRUE;
   FP_SIM.WORK.CON1 := TRUE;
   FP_SIM.WORK.RES := TRUE;
   AdapterBlock.Intell_Type := 54;
   AdapterBlock.VersionNo := 420;
   AdapterBlock.BuildNo := 1;
   AdapterBlock.FuncType := 41;
   AdapterBlock.NetNo := 105;
   AdapterBlock.NodeNo := 42;
   AdapterBlock.Flash_Slow := TRUE;
   AdapterBlock.CON1 := TRUE;
   AdapterBlock.RES := TRUE;
   AdapterBlock.HMI_BOOL[3] := TRUE;
   AdapterBlock.HMI_BOOL[4] := TRUE;
   AdapterBlock.HMI_BOOL[8] := TRUE;
   AdapterBlock.HMI_BOOL[20] := TRUE;
   AdapterBlock.HMI_BOOL[25] := TRUE;
   AdapterBlock.HMI_BOOL[28] := TRUE;
   AdapterBlock.HMI_BOOL[74] := TRUE;
   STATE.A_Running1 := TRUE;
   ONS.Unimotor := TRUE;
   ONS.MD_OnOff := TRUE;
   ONS.Cmd_Auto := TRUE;
   ONS.GLTP := TRUE;
   ONS.RET1 := TRUE;
   ONS.MD_Pulse := TRUE;
   ONS.CMD_Start1 := TRUE;
   ONS.CMD_Start2 := TRUE;
   ONS.SecPulse1 := TRUE;
   StatusWork := 81;
   ModePointer := 51;
   StartWarn_Mem := 15;
   DelayStop_Mem := 5;
   ReturnMon_Mem := 2;
   SpeedMonOnDelay_Mem := 10;
   SpeedMonOffDelay_Mem := 10;
   LeaveFS_Mem := 5;
   ReachLS_Mem := 30;
   ReachFS_Mem := 10;
   ModeAuto := TRUE;
   Select := TRUE;
   FromStateAuto := TRUE;
   Rundelay1_Done := TRUE;
   ChangeDir2_Done := TRUE;
   RET1_OneScan := TRUE;
   OUT.CON1 := TRUE;
   OUT.LAMP1 := TRUE;
   OUT.SACK := TRUE;
   OUT.RD1 := TRUE;
   OUT.RUN1 := TRUE;
   OUT.OK := TRUE;
   OUT.AUT := TRUE;
   OUT.RES := TRUE;
   OUT.INTL_OK_STAT := TRUE;
   OUT.INTL_SEQ_STR1_OK_STAT := TRUE;
   OUT.INTL_SEQ_STR2_OK_STAT := TRUE;
   MSW_Status_Trans := 4177;
END_DATA_BLOCK

DATA_BLOCK "_2010BF110U01_DB"   // DB4011
TITLE = Instance DB Unimotor: _2010BF110U01 Feeder
{ S7_Optimized_Access := 'FALSE' }
AUTHOR : METIS
NAME : UNIMO_DB
VERSION : 8.0
// stored: InstanceOfName ACESYS_MOTOR
"ACESYS_MOTOR"
BEGIN
   FP_SEL.MD_OnOff := TRUE;
   FP_SEL.STW_Local := TRUE;
   FP_SEL.STW_Manual := TRUE;
   FP_SEL.STW_Single := TRUE;
   FP_SEL.Type_Unimotor := TRUE;
   FP_SEL.ParentCollection := TRUE;
   FP_EN.Mode_Auto := TRUE;
   FP_EN.Mode_Man := TRUE;
   FP_EN.PB_QStop := TRUE;
   FP_SHOW.AI1 := TRUE;
   FP_SHOW.OVL := TRUE;
   FP_SHOW.DRDY := TRUE;
   FP_SHOW.GFA := TRUE;
   FP_SHOW.BUSF := TRUE;
   FP_SHOW.ACK := TRUE;
   FP_SHOW.PB_Reset := TRUE;
   FP_PARM.StartWarn_Pre := 15;
   FP_PARM.RunDelay1_Pre := 10;
   FP_PARM.ReturnMon_Pre := 2;
   FP_PARM.SpeedMonOnDelay_Pre := 10;
   FP_PARM.SpeedMonOffDelay_Pre := 10;
   FP_PARM.LeaveFS_Pre := 5;
   FP_PARM.ReachLS_Pre := 30;
   FP_PARM.ReachFS_Pre := 10;
   FP_PARM.AI1_Max := 139.0;
   FP_PARM.AI2_Max := 100.0;
   FP_PARM.AI3_Max := 100.0;
   FP_PARM.AO1a_Max := 100.0;
   FP_PARM.AO2a_Max := 100.0;
   FP_PARM.AO3a_Max := 100.0;
   FP_PARM.AO1b_Max := 139.0;
   FP_PARM.AO2b_Max := 75.0;
   FP_PARM.AO3b_Max := 945.0;
   CMD.GSEL := TRUE;
   RET1 := TRUE;
   MD := FALSE;
   SFS := FALSE;
   ES := TRUE;
   AI1 := 125.5;
   AI2 := 404.3;
   AI3 := 30.0;
   SPSET := 30.0;
   INTL.OK := TRUE;
   INTL.DetectFirst := TRUE;
   INTL.ClearFirst := TRUE;
   INTL_SEQ_STR1.OK := TRUE;
   INTL_SEQ_STR1.DetectFirst := TRUE;
   INTL_SEQ_STR1.ClearFirst := TRUE;
   INTL_SEQ_STR2.OK := TRUE;
   INTL_SEQ_STR2.ClearFirst := TRUE;
   INTL_SEQ_STP.OK := TRUE;
   CON1 := TRUE;
   LAMP1 := TRUE;
   SACK := TRUE;
   RD1 := TRUE;
   RUN1 := TRUE;
   OK := TRUE;
   AUT := TRUE;
   AO1a := 90.28777;
   AO1b := 125.5;
   AO2a := 404.3;
   AO2b := 303.225;
   AO3a := 30.0;
   AO3b := 283.5;
   CV := 30.0;
   MSW.EXT.Operation := TRUE;
   MSW.Status := 4177;
   MSW.TimeStamp := 16#3D72;
   BlockInfo.Ace_Version := 80;
   BlockInfo.Ace_BuildNo := 13;
   BlockInfo.State_Act := 108;
   BlockInfo.State_Prev := 106;
   BlockInfo.DB_Number := 4011;
   FP_CMD.Auto := TRUE;
   FP_DIM.Reset := TRUE;
   FP_SHOW.PB_Auto := TRUE;
   FP_SHOW.PB_Manual := TRUE;
   FP_SHOW.PB_Start1 := TRUE;
   FP_SHOW.PB_Stop := TRUE;
   FP_SHOW.AI2 := TRUE;
   FP_SHOW.AI3 := TRUE;
   FP_SHOW.SP := TRUE;
   FP_PARM.StartWarn_Acc := 15;
   FP_PARM.RunDelay1_Acc := 10;
   FP_PARM.ReturnMon_Acc := 2;
   FP_PARM.SpeedMonOnDelay_Acc := 10;
   FP_PARM.SpeedMonOffDelay_Acc := 10;
   FP_PARM.LeaveFS_Acc := 5;
   FP_PARM.ReachLS_Acc := 30;
   FP_PARM.ReachFS_Acc := 10;
   FP_PARM.MD_Freq_SP := 1;
   FP_PARM.INTL := TRUE;
   FP_PARM.INTL_SEQ_STR1 := TRUE;
   FP_PARM.INTL_SEQ_STR2 := TRUE;
   FP_PARM.INTL_SEQ_STP := TRUE;
   FP_SIM.OVL_Enable := TRUE;
   FP_SIM.RDY_Enable := TRUE;
   FP_SIM.SSW_Enable := TRUE;
   FP_SIM.TFA_Enable := TRUE;
   FP_SIM.MCC_Enable := TRUE;
   FP_SIM.DRDY_Enable := TRUE;
   FP_SIM.MD_Enable := TRUE;
   FP_SIM.GFA_Enable := TRUE;
   FP_SIM.GWA_Enable := TRUE;
   FP_SIM.STALL_Enable := TRUE;
   FP_SIM.EARTH_Enable := TRUE;
   FP_SIM.UBAL_Enable := TRUE;
   FP_SIM.BUSF_Enable := TRUE;
   FP_SIM.RET1_Enable := TRUE;
   FP_SIM.RET2_Enable := TRUE;
   FP_SIM.DOPR_Enable := TRUE;
   FP_SIM.ACK_Enable := TRUE;
   FP_SIM.LSTP_Enable := TRUE;
   FP_SIM.REM_Enable := TRUE;
   FP_SIM.SFS_Enable := TRUE;
   FP_SIM.SLS_Enable := TRUE;
   FP_SIM.ES_Enable := TRUE;
   FP_SIM.WORK.Flash_Slow := TRUE;
   FP_SIM.WORK.CON1 := TRUE;
   AdapterBlock.Intell_Type := 333;
   AdapterBlock.VersionNo := 1;
   AdapterBlock.Flash_Slow := TRUE;
   AdapterBlock.Flash_Fast := TRUE;
   AdapterBlock.CON1 := TRUE;
   AdapterBlock.HMI_INT[1] := 150;
   AdapterBlock.HMI_INT[4] := 500;
   AdapterBlock.HMI_INT[7] := 150;
   AdapterBlock.HMI_INT[9] := 1591;
   AdapterBlock.HMI_INT[11] := 1;
   AdapterBlock.HMI_REAL[1] := 30.0;
   AdapterBlock.HMI_REAL[4] := 125.5;
   AdapterBlock.HMI_REAL[8] := 100.0;
   AdapterBlock.HMI_REAL[13] := 1255.0;
   AdapterBlock.HMI_BOOL[3] := TRUE;
   AdapterBlock.HMI_BOOL[4] := TRUE;
   AdapterBlock.HMI_BOOL[8] := TRUE;
   AdapterBlock.HMI_BOOL[20] := TRUE;
   AdapterBlock.HMI_BOOL[25] := TRUE;
   AdapterBlock.HMI_BOOL[28] := TRUE;
   STATE.A_Running1 := TRUE;
   ONS.Unimotor := TRUE;
   ONS.MD_OnOff := TRUE;
   ONS.Cmd_Auto := TRUE;
   ONS.GLTP := TRUE;
   ONS.RET1 := TRUE;
   ONS.CMD_Start1 := TRUE;
   ONS.CMD_Start2 := TRUE;
   ONS.SecPulse1 := TRUE;
   StatusWork := 81;
   ModePointer := 51;
   StartWarn_Mem := 15;
   ReturnMon_Mem := 2;
   SpeedMonOnDelay_Mem := 10;
   SpeedMonOffDelay_Mem := 10;
   LeaveFS_Mem := 5;
   ReachLS_Mem := 30;
   ReachFS_Mem := 10;
   ModeAuto := TRUE;
   Select := TRUE;
   FromStateAuto := TRUE;
   Rundelay1_Done := TRUE;
   ChangeDir2_Done := TRUE;
   RET1_OneScan := TRUE;
   OUT.CON1 := TRUE;
   OUT.LAMP1 := TRUE;
   OUT.SACK := TRUE;
   OUT.RD1 := TRUE;
   OUT.RUN1 := TRUE;
   OUT.OK := TRUE;
   OUT.AUT := TRUE;
   OUT.INTL_OK_STAT := TRUE;
   OUT.INTL_SEQ_STR1_OK_STAT := TRUE;
   OUT.INTL_SEQ_STR2_OK_STAT := TRUE;
   OUT.INTL_SEQ_STP_OK_STAT := TRUE;
   MSW_Status_Trans := 4177;
END_DATA_BLOCK

DATA_BLOCK "_2010SC130U01_DB"   // DB4012
TITLE = Instance DB Unimotor: _2010SC130U01 Screen
{ S7_Optimized_Access := 'FALSE' }
AUTHOR : METIS
NAME : UNIMO_DB
VERSION : 8.0
// stored: InstanceOfName ACESYS_MOTOR
"ACESYS_MOTOR"
BEGIN
   FP_SEL.MD_OnOff := TRUE;
   FP_SEL.STW_Manual := TRUE;
   FP_SEL.STW_Single := TRUE;
   FP_SEL.Type_Unimotor := TRUE;
   FP_SEL.ParentCollection := TRUE;
   FP_EN.Mode_Auto := TRUE;
   FP_EN.Mode_Man := TRUE;
   FP_EN.PB_QStop := TRUE;
   FP_SHOW.AI1 := TRUE;
   FP_SHOW.OVL := TRUE;
   FP_SHOW.DRDY := TRUE;
   FP_SHOW.STALL := TRUE;
   FP_SHOW.EARTH := TRUE;
   FP_SHOW.GFA := TRUE;
   FP_SHOW.BUSF := TRUE;
   FP_SHOW.ACK := TRUE;
   FP_SHOW.PB_Reset := TRUE;
   FP_PARM.StartWarn_Pre := 15;
   FP_PARM.RunDelay1_Pre := 5;
   FP_PARM.DelayStop_Pre := 5;
   FP_PARM.ReturnMon_Pre := 30;
   FP_PARM.SpeedMonOnDelay_Pre := 10;
   FP_PARM.SpeedMonOffDelay_Pre := 10;
   FP_PARM.LeaveFS_Pre := 5;
   FP_PARM.ReachLS_Pre := 30;
   FP_PARM.ReachFS_Pre := 10;
   FP_PARM.AI1_Max := 134.0;
   FP_PARM.AI2_Max := 100.0;
   FP_PARM.AI3_Max := 100.0;
   FP_PARM.AO1a_Max := 100.0;
   FP_PARM.AO2a_Max := 100.0;
   FP_PARM.AO3a_Max := 100.0;
   FP_PARM.AO1b_Max := 134.0;
   FP_PARM.AO2b_Max := 75.0;
   FP_PARM.AO3b_Max := 1485.0;
   CMD.GSEL := TRUE;
   RET1 := TRUE;
   MD := FALSE;
   SFS := FALSE;
   ES := TRUE;
   AI1 := 49.7;
   AI2 := 406.1;
   AI3 := 100.0;
   SPSET := 100.0;
   INTL.OK := TRUE;
   INTL.DetectFirst := TRUE;
   INTL.ClearFirst := TRUE;
   INTL_SEQ_STR1.OK := TRUE;
   INTL_SEQ_STR1.DetectFirst := TRUE;
   INTL_SEQ_STR1.ClearFirst := TRUE;
   INTL_SEQ_STR2.OK := TRUE;
   INTL_SEQ_STR2.ClearFirst := TRUE;
   INTL_SEQ_STP.OK := TRUE;
   CON1 := TRUE;
   LAMP1 := TRUE;
   SACK := TRUE;
   RD1 := TRUE;
   RUN1 := TRUE;
   OK := TRUE;
   AUT := TRUE;
   AO1a := 37.08955;
   AO1b := 49.7;
   AO2a := 406.1;
   AO2b := 304.575;
   AO3a := 100.0;
   AO3b := 1485.0;
   CV := 100.0;
   MSW.EXT.Operation := TRUE;
   MSW.Status := 4177;
   MSW.TimeStamp := 16#353D;
   BlockInfo.Ace_Version := 80;
   BlockInfo.Ace_BuildNo := 13;
   BlockInfo.State_Act := 108;
   BlockInfo.State_Prev := 106;
   BlockInfo.DB_Number := 4012;
   FP_CMD.Auto := TRUE;
   FP_DIM.Reset := TRUE;
   FP_SHOW.PB_Auto := TRUE;
   FP_SHOW.PB_Manual := TRUE;
   FP_SHOW.PB_Start1 := TRUE;
   FP_SHOW.PB_Stop := TRUE;
   FP_SHOW.AI2 := TRUE;
   FP_SHOW.AI3 := TRUE;
   FP_SHOW.SP := TRUE;
   FP_PARM.StartWarn_Acc := 15;
   FP_PARM.RunDelay1_Acc := 5;
   FP_PARM.DelayStop_Acc := 5;
   FP_PARM.ReturnMon_Acc := 30;
   FP_PARM.SpeedMonOnDelay_Acc := 10;
   FP_PARM.SpeedMonOffDelay_Acc := 10;
   FP_PARM.LeaveFS_Acc := 5;
   FP_PARM.ReachLS_Acc := 30;
   FP_PARM.ReachFS_Acc := 10;
   FP_PARM.MD_Freq_SP := 1;
   FP_PARM.INTL := TRUE;
   FP_PARM.INTL_SEQ_STR1 := TRUE;
   FP_PARM.INTL_SEQ_STR2 := TRUE;
   FP_SIM.OVL_Enable := TRUE;
   FP_SIM.RDY_Enable := TRUE;
   FP_SIM.SSW_Enable := TRUE;
   FP_SIM.TFA_Enable := TRUE;
   FP_SIM.MCC_Enable := TRUE;
   FP_SIM.DRDY_Enable := TRUE;
   FP_SIM.MD_Enable := TRUE;
   FP_SIM.GFA_Enable := TRUE;
   FP_SIM.GWA_Enable := TRUE;
   FP_SIM.STALL_Enable := TRUE;
   FP_SIM.EARTH_Enable := TRUE;
   FP_SIM.UBAL_Enable := TRUE;
   FP_SIM.BUSF_Enable := TRUE;
   FP_SIM.RET1_Enable := TRUE;
   FP_SIM.RET2_Enable := TRUE;
   FP_SIM.DOPR_Enable := TRUE;
   FP_SIM.ACK_Enable := TRUE;
   FP_SIM.LSTP_Enable := TRUE;
   FP_SIM.REM_Enable := TRUE;
   FP_SIM.SFS_Enable := TRUE;
   FP_SIM.SLS_Enable := TRUE;
   FP_SIM.ES_Enable := TRUE;
   FP_SIM.WORK.Flash_Slow := TRUE;
   FP_SIM.WORK.CON1 := TRUE;
   AdapterBlock.Intell_Type := 333;
   AdapterBlock.VersionNo := 1;
   AdapterBlock.Flash_Slow := TRUE;
   AdapterBlock.Flash_Fast := TRUE;
   AdapterBlock.CON1 := TRUE;
   AdapterBlock.HMI_INT[1] := 500;
   AdapterBlock.HMI_INT[4] := 500;
   AdapterBlock.HMI_INT[7] := 500;
   AdapterBlock.HMI_INT[9] := 1591;
   AdapterBlock.HMI_INT[11] := 1;
   AdapterBlock.HMI_REAL[1] := 100.0;
   AdapterBlock.HMI_REAL[4] := 49.7;
   AdapterBlock.HMI_REAL[8] := 100.0;
   AdapterBlock.HMI_REAL[13] := 497.0;
   AdapterBlock.HMI_BOOL[3] := TRUE;
   AdapterBlock.HMI_BOOL[4] := TRUE;
   AdapterBlock.HMI_BOOL[8] := TRUE;
   AdapterBlock.HMI_BOOL[20] := TRUE;
   AdapterBlock.HMI_BOOL[25] := TRUE;
   AdapterBlock.HMI_BOOL[28] := TRUE;
   STATE.A_Running1 := TRUE;
   ONS.Unimotor := TRUE;
   ONS.MD_OnOff := TRUE;
   ONS.Cmd_Auto := TRUE;
   ONS.GLTP := TRUE;
   ONS.RET1 := TRUE;
   ONS.CMD_Start1 := TRUE;
   ONS.CMD_Start2 := TRUE;
   ONS.SecPulse1 := TRUE;
   StatusWork := 81;
   ModePointer := 51;
   StartWarn_Mem := 15;
   DelayStop_Mem := 5;
   ReturnMon_Mem := 30;
   SpeedMonOnDelay_Mem := 10;
   SpeedMonOffDelay_Mem := 10;
   LeaveFS_Mem := 5;
   ReachLS_Mem := 30;
   ReachFS_Mem := 10;
   ModeAuto := TRUE;
   Select := TRUE;
   FromStateAuto := TRUE;
   Rundelay1_Done := TRUE;
   ChangeDir2_Done := TRUE;
   RET1_OneScan := TRUE;
   OUT.CON1 := TRUE;
   OUT.LAMP1 := TRUE;
   OUT.SACK := TRUE;
   OUT.RD1 := TRUE;
   OUT.RUN1 := TRUE;
   OUT.OK := TRUE;
   OUT.AUT := TRUE;
   OUT.INTL_OK_STAT := TRUE;
   OUT.INTL_SEQ_STR1_OK_STAT := TRUE;
   OUT.INTL_SEQ_STR2_OK_STAT := TRUE;
   MSW_Status_Trans := 4177;
END_DATA_BLOCK

DATA_BLOCK "_2010CR150M01_DB"   // DB4013
TITLE = Instance DB Unimotor: Crusher CR150
{ S7_Optimized_Access := 'FALSE' }
AUTHOR : METIS
NAME : UNIMO_DB
VERSION : 8.0
// stored: InstanceOfName ACESYS_MOTOR
"ACESYS_MOTOR"
BEGIN
   FP_SEL.MD_OnOff := TRUE;
   FP_SEL.STW_Local := TRUE;
   FP_SEL.STW_Manual := TRUE;
   FP_SEL.STW_Single := TRUE;
   FP_SEL.Type_Unimotor := TRUE;
   FP_SEL.ParentSupress := TRUE;
   FP_SEL.ParentCollection := TRUE;
   FP_EN.Mode_Auto := TRUE;
   FP_EN.Mode_Man := TRUE;
   FP_EN.PB_QStop := TRUE;
   FP_SHOW.AI1 := TRUE;
   FP_SHOW.DRDY := TRUE;
   FP_SHOW.GFA := TRUE;
   FP_SHOW.PB_Reset := TRUE;
   FP_PARM.StartWarn_Pre := 15;
   FP_PARM.RunDelay1_Pre := 5;
   FP_PARM.DelayStop_Pre := 30;
   FP_PARM.ReturnMon_Pre := 2;
   FP_PARM.SpeedMonOnDelay_Pre := 10;
   FP_PARM.SpeedMonOffDelay_Pre := 10;
   FP_PARM.LeaveFS_Pre := 5;
   FP_PARM.ReachLS_Pre := 30;
   FP_PARM.ReachFS_Pre := 10;
   FP_PARM.AI1_Max := 435.0;
   FP_PARM.AI2_Max := 100.0;
   FP_PARM.AI3_Max := 100.0;
   FP_PARM.AO1a_Max := 100.0;
   FP_PARM.AO2a_Max := 100.0;
   FP_PARM.AO3a_Max := 100.0;
   FP_PARM.AO1b_Max := 435.0;
   FP_PARM.AO2b_Max := 100.0;
   FP_PARM.AO3b_Max := 100.0;
   CMD.GSEL := TRUE;
   RET1 := TRUE;
   MD := FALSE;
   SFS := FALSE;
   ES := TRUE;
   AI1 := 6.741643;
   INTL.OK := TRUE;
   INTL.DetectFirst := TRUE;
   INTL.ClearFirst := TRUE;
   INTL_SEQ_STR1.OK := TRUE;
   INTL_SEQ_STR1.DetectFirst := TRUE;
   INTL_SEQ_STR1.ClearFirst := TRUE;
   INTL_SEQ_STR2.OK := TRUE;
   INTL_SEQ_STR2.ClearFirst := TRUE;
   INTL_SEQ_STP.OK := TRUE;
   CON1 := TRUE;
   LAMP1 := TRUE;
   SACK := TRUE;
   RD1 := TRUE;
   RUN1 := TRUE;
   OK := TRUE;
   AUT := TRUE;
   RES := TRUE;
   AO1a := 1.549803;
   AO1b := 6.741643;
   MSW.EXT.Operation := TRUE;
   MSW.Status := 4177;
   MSW.TimeStamp := 16#82ED;
   BlockInfo.Ace_Version := 80;
   BlockInfo.Ace_BuildNo := 13;
   BlockInfo.State_Act := 108;
   BlockInfo.State_Prev := 106;
   BlockInfo.DB_Number := 4013;
   FP_CMD.Auto := TRUE;
   FP_DIM.Reset := TRUE;
   FP_SHOW.PB_Auto := TRUE;
   FP_SHOW.PB_Manual := TRUE;
   FP_SHOW.PB_Start1 := TRUE;
   FP_SHOW.PB_Stop := TRUE;
   FP_PARM.StartWarn_Acc := 15;
   FP_PARM.RunDelay1_Acc := 5;
   FP_PARM.DelayStart_Pre := 10;
   FP_PARM.DelayStart_Acc := 10;
   FP_PARM.DelayStop_Acc := 30;
   FP_PARM.ReturnMon_Acc := 2;
   FP_PARM.SpeedMonOnDelay_Acc := 10;
   FP_PARM.SpeedMonOffDelay_Acc := 10;
   FP_PARM.LeaveFS_Acc := 5;
   FP_PARM.ReachLS_Acc := 30;
   FP_PARM.ReachFS_Acc := 10;
   FP_PARM.MD_Freq_SP := 1;
   FP_PARM.INTL := TRUE;
   FP_PARM.INTL_SEQ_STR1 := TRUE;
   FP_PARM.INTL_SEQ_STR2 := TRUE;
   FP_PARM.INTL_SEQ_STP := TRUE;
   FP_SIM.OVL_Enable := TRUE;
   FP_SIM.RDY_Enable := TRUE;
   FP_SIM.SSW_Enable := TRUE;
   FP_SIM.TFA_Enable := TRUE;
   FP_SIM.MCC_Enable := TRUE;
   FP_SIM.DRDY_Enable := TRUE;
   FP_SIM.MD_Enable := TRUE;
   FP_SIM.GFA_Enable := TRUE;
   FP_SIM.GWA_Enable := TRUE;
   FP_SIM.STALL_Enable := TRUE;
   FP_SIM.EARTH_Enable := TRUE;
   FP_SIM.UBAL_Enable := TRUE;
   FP_SIM.BUSF_Enable := TRUE;
   FP_SIM.RET1_Enable := TRUE;
   FP_SIM.RET2_Enable := TRUE;
   FP_SIM.DOPR_Enable := TRUE;
   FP_SIM.ACK_Enable := TRUE;
   FP_SIM.LSTP_Enable := TRUE;
   FP_SIM.REM_Enable := TRUE;
   FP_SIM.SFS_Enable := TRUE;
   FP_SIM.SLS_Enable := TRUE;
   FP_SIM.ES_Enable := TRUE;
   FP_SIM.WORK.Flash_Slow := TRUE;
   FP_SIM.WORK.CON1 := TRUE;
   FP_SIM.WORK.RES := TRUE;
   AdapterBlock.Intell_Type := 54;
   AdapterBlock.VersionNo := 420;
   AdapterBlock.BuildNo := 1;
   AdapterBlock.FuncType := 41;
   AdapterBlock.NetNo := 105;
   AdapterBlock.NodeNo := 42;
   AdapterBlock.Flash_Slow := TRUE;
   AdapterBlock.Flash_Fast := TRUE;
   AdapterBlock.CON1 := TRUE;
   AdapterBlock.RES := TRUE;
   AdapterBlock.HMI_BOOL[3] := TRUE;
   AdapterBlock.HMI_BOOL[4] := TRUE;
   AdapterBlock.HMI_BOOL[8] := TRUE;
   AdapterBlock.HMI_BOOL[20] := TRUE;
   AdapterBlock.HMI_BOOL[25] := TRUE;
   AdapterBlock.HMI_BOOL[28] := TRUE;
   AdapterBlock.HMI_BOOL[74] := TRUE;
   STATE.A_Running1 := TRUE;
   ONS.Unimotor := TRUE;
   ONS.MD_OnOff := TRUE;
   ONS.Cmd_Auto := TRUE;
   ONS.GLTP := TRUE;
   ONS.RET1 := TRUE;
   ONS.CMD_Start1 := TRUE;
   ONS.CMD_Start2 := TRUE;
   ONS.SecPulse1 := TRUE;
   StatusWork := 81;
   ModePointer := 51;
   StartWarn_Mem := 15;
   DelayStart_Mem := 10;
   DelayStop_Mem := 30;
   ReturnMon_Mem := 2;
   SpeedMonOnDelay_Mem := 10;
   SpeedMonOffDelay_Mem := 10;
   LeaveFS_Mem := 5;
   ReachLS_Mem := 30;
   ReachFS_Mem := 10;
   ModeAuto := TRUE;
   Select := TRUE;
   FromStateAuto := TRUE;
   Rundelay1_Done := TRUE;
   ChangeDir2_Done := TRUE;
   RET1_OneScan := TRUE;
   OUT.CON1 := TRUE;
   OUT.LAMP1 := TRUE;
   OUT.SACK := TRUE;
   OUT.RD1 := TRUE;
   OUT.RUN1 := TRUE;
   OUT.OK := TRUE;
   OUT.AUT := TRUE;
   OUT.RES := TRUE;
   OUT.INTL_OK_STAT := TRUE;
   OUT.INTL_SEQ_STR1_OK_STAT := TRUE;
   OUT.INTL_SEQ_STR2_OK_STAT := TRUE;
   OUT.INTL_SEQ_STP_OK_STAT := TRUE;
   MSW_Status_Trans := 4177;
END_DATA_BLOCK

DATA_BLOCK "_2010SJ950M01_DB"   // DB4110
TITLE = Instance DB Unimotor: _2010SJ950M01
{ S7_Optimized_Access := 'FALSE' }
AUTHOR : METIS
NAME : UNIMO_DB
VERSION : 8.0
// stored: InstanceOfName ACESYS_MOTOR
"ACESYS_MOTOR"
BEGIN
   FP_SEL.MD_OnOff := TRUE;
   FP_SEL.STW_Local := TRUE;
   FP_SEL.STW_Manual := TRUE;
   FP_SEL.STW_Single := TRUE;
   FP_SEL.Type_Unimotor := TRUE;
   FP_SEL.ParentSupress := TRUE;
   FP_SEL.ParentCollection := TRUE;
   FP_EN.Mode_Auto := TRUE;
   FP_EN.Mode_Man := TRUE;
   FP_EN.Mode_Loc := TRUE;
   FP_EN.Mode_SS_Field := TRUE;
   FP_EN.Mode_SS_FP := TRUE;
   FP_EN.PB_QStop := TRUE;
   FP_SHOW.AI1 := TRUE;
   FP_SHOW.OVL := TRUE;
   FP_SHOW.LSTP := TRUE;
   FP_SHOW.DRDY := TRUE;
   FP_SHOW.STALL := TRUE;
   FP_SHOW.EARTH := TRUE;
   FP_SHOW.UBAL := TRUE;
   FP_SHOW.GFA := TRUE;
   FP_SHOW.GWA := TRUE;
   FP_SHOW.BUSF := TRUE;
   FP_SHOW.DOPR := TRUE;
   FP_SHOW.DTEST := TRUE;
   FP_SHOW.ACK := TRUE;
   FP_SHOW.PB_Reset := TRUE;
   FP_SHOW.ASTR := TRUE;
   FP_PARM.StartWarn_Pre := 15;
   FP_PARM.RunDelay1_Pre := 5;
   FP_PARM.DelayStop_Pre := 5;
   FP_PARM.ReturnMon_Pre := 2;
   FP_PARM.SpeedMonOnDelay_Pre := 10;
   FP_PARM.SpeedMonOffDelay_Pre := 10;
   FP_PARM.LeaveFS_Pre := 5;
   FP_PARM.ReachLS_Pre := 30;
   FP_PARM.ReachFS_Pre := 10;
   FP_PARM.AI1_Max := 100.0;
   FP_PARM.AI2_Max := 100.0;
   FP_PARM.AI3_Max := 100.0;
   FP_PARM.AO1a_Max := 100.0;
   FP_PARM.AO2a_Max := 100.0;
   FP_PARM.AO3a_Max := 100.0;
   FP_PARM.AO1b_Max := 100.0;
   FP_PARM.AO2b_Max := 100.0;
   FP_PARM.AO3b_Max := 100.0;
   CMD.GSEL := TRUE;
   SEL := FALSE;
   ASTR := FALSE;
   LSTP := FALSE;
   DRDY := FALSE;
   MD := FALSE;
   GFA := FALSE;
   BUSF := FALSE;
   DOPR := FALSE;
   DTEST := TRUE;
   SFS := FALSE;
   ES := TRUE;
   INTL.OK := TRUE;
   INTL_SEQ_STR1.OK := TRUE;
   INTL_SEQ_STR2.OK := TRUE;
   INTL_SEQ_STP.OK := TRUE;
   LAMP1 := TRUE;
   LAMP2 := TRUE;
   AUT := TRUE;
   RES := TRUE;
   AL_SUPR := TRUE;
   MSW.EXT.AlarmSuppressed := TRUE;
   MSW.EXT.AlarmPresent := TRUE;
   MSW.EXT.AlarmFailUnAck := TRUE;
   MSW.Status := 201;
   MSW.TimeStamp := 16#D059;
   BlockInfo.Ace_Version := 80;
   BlockInfo.Ace_BuildNo := 13;
   BlockInfo.State_Act := 607;
   BlockInfo.State_Prev := 101;
   BlockInfo.DB_Number := 4110;
   FP_CMD.Auto := TRUE;
   FP_DIM.Local := TRUE;
   FP_DIM.Manual := TRUE;
   FP_DIM.Reset := TRUE;
   FP_SHOW.PB_Auto := TRUE;
   FP_SHOW.PB_Local := TRUE;
   FP_SHOW.PB_Manual := TRUE;
   FP_SHOW.PB_Start1 := TRUE;
   FP_SHOW.PB_Stop := TRUE;
   FP_SHOW.LSTR1 := TRUE;
   FP_PARM.StartWarn_Acc := 15;
   FP_PARM.RunDelay1_Acc := 5;
   FP_PARM.DelayStop_Acc := 5;
   FP_PARM.ReturnMon_Acc := 2;
   FP_PARM.SpeedMonOnDelay_Acc := 10;
   FP_PARM.SpeedMonOffDelay_Acc := 10;
   FP_PARM.LeaveFS_Acc := 5;
   FP_PARM.ReachLS_Acc := 30;
   FP_PARM.ReachFS_Acc := 10;
   FP_PARM.MD_Freq_SP := 1;
   FP_PARM.StopReason := 10;
   FP_PARM.INTL := TRUE;
   FP_PARM.INTL_SEQ_STR2 := TRUE;
   FP_PARM.INTL_SEQ_STP := TRUE;
   FP_SIM.OVL_Enable := TRUE;
   FP_SIM.RDY_Enable := TRUE;
   FP_SIM.SSW_Enable := TRUE;
   FP_SIM.TFA_Enable := TRUE;
   FP_SIM.MCC_Enable := TRUE;
   FP_SIM.DRDY_Enable := TRUE;
   FP_SIM.MD_Enable := TRUE;
   FP_SIM.GFA_Enable := TRUE;
   FP_SIM.GWA_Enable := TRUE;
   FP_SIM.STALL_Enable := TRUE;
   FP_SIM.EARTH_Enable := TRUE;
   FP_SIM.UBAL_Enable := TRUE;
   FP_SIM.BUSF_Enable := TRUE;
   FP_SIM.RET1_Enable := TRUE;
   FP_SIM.RET2_Enable := TRUE;
   FP_SIM.DOPR_Enable := TRUE;
   FP_SIM.ACK_Enable := TRUE;
   FP_SIM.LSTP_Enable := TRUE;
   FP_SIM.REM_Enable := TRUE;
   FP_SIM.SFS_Enable := TRUE;
   FP_SIM.SLS_Enable := TRUE;
   FP_SIM.ES_Enable := TRUE;
   FP_SIM.WORK.Flash_Slow := TRUE;
   FP_SIM.WORK.RES := TRUE;
   AdapterBlock.Intell_Type := 54;
   AdapterBlock.VersionNo := 420;
   AdapterBlock.BuildNo := 1;
   AdapterBlock.FuncType := 41;
   AdapterBlock.NetNo := 106;
   AdapterBlock.NodeNo := 26;
   AdapterBlock.Flash_Slow := TRUE;
   AdapterBlock.RES := TRUE;
   AdapterBlock.HMI_BOOL[3] := TRUE;
   AdapterBlock.HMI_BOOL[4] := TRUE;
   AdapterBlock.HMI_BOOL[8] := TRUE;
   AdapterBlock.HMI_BOOL[74] := TRUE;
   STATE.Alarm := TRUE;
   ONS.Unimotor := TRUE;
   ONS.MD_OnOff := TRUE;
   ONS.Cmd_Auto := TRUE;
   ONS.GLTP := TRUE;
   ONS.CMD_Start1 := TRUE;
   ONS.CMD_Start2 := TRUE;
   ONS.SecPulse2 := TRUE;
   StatusWork := 201;
   ModePointer := 51;
   AlarmNo := 23;
   AlarmNo_Old := 23;
   StartWarn_Mem := 15;
   RunDelay1_Mem := 5;
   DelayStop_Mem := 5;
   ReturnMon_Mem := 2;
   SpeedMonOnDelay_Mem := 10;
   SpeedMonOffDelay_Mem := 10;
   LeaveFS_Mem := 5;
   ReachLS_Mem := 30;
   ReachFS_Mem := 10;
   ModeAuto := TRUE;
   FromStopState := TRUE;
   ALARM_SupressionActive := TRUE;
   ALARM_AlarmPresent := TRUE;
   ChangeDir1_Done := TRUE;
   ChangeDir2_Done := TRUE;
   OUT.LAMP1 := TRUE;
   OUT.LAMP2 := TRUE;
   OUT.AUT := TRUE;
   OUT.RES := TRUE;
   OUT.AL_SUPR := TRUE;
   OUT.INTL_OK_STAT := TRUE;
   OUT.INTL_SEQ_STR2_OK_STAT := TRUE;
   OUT.INTL_SEQ_STP_OK_STAT := TRUE;
   MSW_Status_Trans := 201;
END_DATA_BLOCK

DATA_BLOCK "_2090TK730Y01_DB"   // DB4169
{ S7_Optimized_Access := 'FALSE' }
AUTHOR : FLSmidth
FAMILY : ACESYS
NAME : VALVE
VERSION : 8.0
// stored: InstanceOfName ACESYS_VALVE
"ACESYS_VALVE"
BEGIN
   FP_SIM.OVL_Enable := TRUE;
   FP_SIM.RDY_Enable := TRUE;
   FP_SIM.SSW_Enable := TRUE;
   FP_SIM.DRDY_Enable := TRUE;
   FP_SIM.GFA_Enable := TRUE;
   FP_SIM.GWA_Enable := TRUE;
   FP_SIM.Spare_Enable := TRUE;
   FP_SIM.BUSF_Enable := TRUE;
   FP_SIM.ACK_Enable := TRUE;
   FP_SIM.REM_Enable := TRUE;
   FP_SIM.LSP1_Enable := TRUE;
   FP_SIM.LSP2_Enable := TRUE;
   FP_SIM.LSP3_Enable := TRUE;
END_DATA_BLOCK

DATA_BLOCK "_2010LV100P01_DB"   // DB4357
TITLE = Instance DB Power Monitor: _2010LV100P01
{ S7_Optimized_Access := 'FALSE' }
AUTHOR : METIS
NAME : POWER_DB
VERSION : 8.0
// stored: InstanceOfName ACESYS_POWER
"ACESYS_POWER"
BEGIN
   MSW.EXT.Operation := TRUE;
   MSW.Status := 1;
   MSW.TimeStamp := 16#0D08;
   BlockInfo.Ace_Version := 80;
   BlockInfo.Ace_BuildNo := 1;
   BlockInfo.DB_Number := 4357;
   FP_SEL.Type_Monitor := TRUE;
   FP_VIS.Power := TRUE;
   FP_VIS.Energy := TRUE;
   LINK.INFO.BuildNo := 1;
   LINK.INFO.NetNo := 106;
   LINK.INFO.NodeNo := 22;
   LINK.INFO.Flash_Slow := TRUE;
   LINK.Status.BUSF := TRUE;
   LINK.Status.HLTY := TRUE;
   LINK.Command.RES := TRUE;
   LINK.EN.VOLT_LNPH := TRUE;
   LINK.EN.CURR_LN := TRUE;
   LINK.EN.APOW_PH := TRUE;
   LINK.EN.FRQ := TRUE;
   LINK.EN.RTPOW_AVG := TRUE;
   LINK.EN.RENG := TRUE;
   LINK.PARM.VOLT_L1L2 := 401.1395;
   LINK.PARM.VOLT_L2L3 := 401.1483;
   LINK.PARM.VOLT_L3L1 := 400.6243;
   LINK.PARM.VOLT_AVG := 400.9707;
   LINK.PARM.CURR_L1 := 176.0122;
   LINK.PARM.CURR_L2 := 183.3011;
   LINK.PARM.CURR_L3 := 179.5082;
   LINK.PARM.CURR_AVG := 179.6072;
   LINK.PARM.FRQ := 49.93077;
   LINK.PARM.PF_AVG := 0.7808338;
   LINK.PARM.APOW_AVG := 124.7373;
   LINK.PARM.RLPOW_AVG := 97.39913;
   LINK.PARM.RTPOW_AVG := 16.73409;
   LINK.PARM.AENG := 300580.6;
   LINK.PARM.RENG := 381756.4;
   Volt_L1N := 231.5914;
   Volt_L2N := 231.5965;
   Volt_L3N := 231.294;
   StatusWork := 1;
   MSW_Status_Trans := 1;
END_DATA_BLOCK

DATA_BLOCK "_2015PU027U01_DB"   // DB4415
TITLE = Instance DB Unimotor:
{ S7_Optimized_Access := 'FALSE' }
AUTHOR : METIS
NAME : UNIMO_DB
VERSION : 8.0
// stored: InstanceOfName ACESYS_MOTOR
"ACESYS_MOTOR"
BEGIN
   FP_SEL.MD_OnOff := TRUE;
   FP_SEL.STW_Local := TRUE;
   FP_SEL.STW_Manual := TRUE;
   FP_SEL.STW_Single := TRUE;
   FP_SEL.Type_Unimotor := TRUE;
   FP_EN.Mode_Auto := TRUE;
   FP_EN.Mode_Man := TRUE;
   FP_EN.Mode_Loc := TRUE;
   FP_EN.Mode_SS_FP := TRUE;
   FP_SHOW.PB_Reset := TRUE;
   FP_PARM.StartWarn_Pre := 15;
   FP_PARM.RunDelay1_Pre := 5;
   FP_PARM.DelayStop_Pre := 5;
   FP_PARM.ReturnMon_Pre := 2;
   FP_PARM.AI1_Max := 10.7;
   FP_PARM.AI2_Max := 100.0;
   FP_PARM.AI3_Max := 100.0;
   FP_PARM.AO1a_Max := 100.0;
   FP_PARM.AO2a_Max := 100.0;
   FP_PARM.AO3a_Max := 100.0;
   FP_PARM.AO1b_Max := 10.7;
   FP_PARM.AO2b_Max := 5.5;
   FP_PARM.AO3b_Max := 100.0;
   SEL := FALSE;
   MD := FALSE;
   SFS := FALSE;
   ES := TRUE;
   INTL.OK := TRUE;
   INTL_SEQ_STR1.OK := TRUE;
   INTL_SEQ_STR2.OK := TRUE;
   INTL_SEQ_STP.OK := TRUE;
   OK := TRUE;
   MAN := TRUE;
   MSW.EXT.ModeBit2 := TRUE;
   MSW.Status := 1;
   MSW.TimeStamp := 16#A8C5;
   BlockInfo.Ace_Version := 80;
   BlockInfo.Ace_BuildNo := 13;
   BlockInfo.State_Act := 300;
   BlockInfo.State_Prev := 305;
   BlockInfo.DB_Number := 4415;
   FP_CMD.Manual := TRUE;
   FP_EN.PB_QStop := TRUE;
   FP_DIM.Auto := TRUE;
   FP_DIM.Local := TRUE;
   FP_DIM.Start1 := TRUE;
   FP_DIM.Start2 := TRUE;
   FP_DIM.Reset := TRUE;
   FP_SHOW.PB_Auto := TRUE;
   FP_SHOW.PB_Local := TRUE;
   FP_SHOW.PB_Manual := TRUE;
   FP_SHOW.PB_Start1 := TRUE;
   FP_SHOW.PB_Stop := TRUE;
   FP_SHOW.AI1 := TRUE;
   FP_SHOW.AI2 := TRUE;
   FP_SHOW.AI3 := TRUE;
   FP_SHOW.SP := TRUE;
   FP_SHOW.OVL := TRUE;
   FP_SHOW.SSW := TRUE;
   FP_SHOW.STALL := TRUE;
   FP_SHOW.EARTH := TRUE;
   FP_SHOW.UBAL := TRUE;
   FP_SHOW.GFA := TRUE;
   FP_SHOW.GWA := TRUE;
   FP_SHOW.BUSF := TRUE;
   FP_SHOW.DOPR := TRUE;
   FP_SHOW.DTEST := TRUE;
   FP_SHOW.LSTR1 := TRUE;
   FP_PARM.StartWarn_Acc := 15;
   FP_PARM.RunDelay1_Acc := 5;
   FP_PARM.DelayStop_Acc := 5;
   FP_PARM.ReturnMon_Acc := 2;
   FP_PARM.MD_Freq_SP := 1;
   FP_PARM.StopReason := 3;
   FP_PARM.INTL := TRUE;
   FP_PARM.INTL_SEQ_STR1 := TRUE;
   FP_PARM.INTL_SEQ_STR2 := TRUE;
   FP_PARM.INTL_SEQ_STP := TRUE;
   FP_SIM.OVL_Enable := TRUE;
   FP_SIM.RDY_Enable := TRUE;
   FP_SIM.SSW_Enable := TRUE;
   FP_SIM.TFA_Enable := TRUE;
   FP_SIM.MCC_Enable := TRUE;
   FP_SIM.DRDY_Enable := TRUE;
   FP_SIM.MD_Enable := TRUE;
   FP_SIM.GFA_Enable := TRUE;
   FP_SIM.GWA_Enable := TRUE;
   FP_SIM.STALL_Enable := TRUE;
   FP_SIM.EARTH_Enable := TRUE;
   FP_SIM.UBAL_Enable := TRUE;
   FP_SIM.BUSF_Enable := TRUE;
   FP_SIM.RET1_Enable := TRUE;
   FP_SIM.RET2_Enable := TRUE;
   FP_SIM.DOPR_Enable := TRUE;
   FP_SIM.ACK_Enable := TRUE;
   FP_SIM.LSTP_Enable := TRUE;
   FP_SIM.REM_Enable := TRUE;
   FP_SIM.SFS_Enable := TRUE;
   FP_SIM.SLS_Enable := TRUE;
   FP_SIM.ES_Enable := TRUE;
   FP_SIM.WORK.Flash_Slow := TRUE;
   AdapterBlock.Intell_Type := 282;
   AdapterBlock.VersionNo := 220;
   AdapterBlock.FuncType := 41;
   AdapterBlock.Options := 1;
   AdapterBlock.NetNo := 106;
   AdapterBlock.NodeNo := 75;
   AdapterBlock.Flash_Slow := TRUE;
   AdapterBlock.Flash_Fast := TRUE;
   AdapterBlock.MAN := TRUE;
   AdapterBlock.HMI_INT[9] := 3;
   AdapterBlock.HMI_INT[10] := 2;
   AdapterBlock.HMI_INT[11] := 6;
   AdapterBlock.HMI_REAL[9] := 100.0;
   AdapterBlock.HMI_REAL[10] := 100.0;
   AdapterBlock.HMI_REAL[12] := 100.0;
   AdapterBlock.HMI_BOOL[1] := TRUE;
   AdapterBlock.HMI_BOOL[2] := TRUE;
   AdapterBlock.HMI_BOOL[9] := TRUE;
   AdapterBlock.HMI_BOOL[15] := TRUE;
   AdapterBlock.HMI_BOOL[17] := TRUE;
   AdapterBlock.HMI_BOOL[18] := TRUE;
   AdapterBlock.HMI_BOOL[34] := TRUE;
   AdapterBlock.HMI_BOOL[35] := TRUE;
   AdapterBlock.HMI_BOOL[65] := TRUE;
   AdapterBlock.HMI_BOOL[89] := TRUE;
   STATE.M_Stopped := TRUE;
   ONS.Unimotor := TRUE;
   ONS.MD_OnOff := TRUE;
   ONS.Cmd_Manual := TRUE;
   ONS.GLTP := TRUE;
   ONS.CMD_Start1 := TRUE;
   ONS.CMD_Start2 := TRUE;
   ONS.SecPulse1 := TRUE;
   StatusWork := 1;
   ModePointer := 52;
   StartWarn_Mem := 15;
   RunDelay1_Mem := 5;
   DelayStop_Mem := 5;
   ReturnMon_Mem := 2;
   ModeManual := TRUE;
   FromStateManual := TRUE;
   ChangeDir1_Done := TRUE;
   ChangeDir2_Done := TRUE;
   OUT.OK := TRUE;
   OUT.MAN := TRUE;
   OUT.INTL_OK_STAT := TRUE;
   OUT.INTL_SEQ_STR1_OK_STAT := TRUE;
   OUT.INTL_SEQ_STR2_OK_STAT := TRUE;
   OUT.INTL_SEQ_STP_OK_STAT := TRUE;
   MSW_Status_Trans := 1;
END_DATA_BLOCK

DATA_BLOCK "_2015PU028U01_DB"   // DB4416
TITLE = Instance DB Unimotor:
{ S7_Optimized_Access := 'FALSE' }
AUTHOR : METIS
NAME : UNIMO_DB
VERSION : 8.0
// stored: InstanceOfName ACESYS_MOTOR
"ACESYS_MOTOR"
BEGIN
   FP_SEL.MD_OnOff := TRUE;
   FP_SEL.STW_Local := TRUE;
   FP_SEL.STW_Manual := TRUE;
   FP_SEL.STW_Single := TRUE;
   FP_SEL.Type_Unimotor := TRUE;
   FP_EN.Mode_Auto := TRUE;
   FP_EN.Mode_Man := TRUE;
   FP_EN.Mode_Loc := TRUE;
   FP_EN.Mode_SS_FP := TRUE;
   FP_SHOW.PB_Reset := TRUE;
   FP_PARM.StartWarn_Pre := 15;
   FP_PARM.RunDelay1_Pre := 5;
   FP_PARM.DelayStop_Pre := 5;
   FP_PARM.ReturnMon_Pre := 2;
   FP_PARM.AI1_Max := 10.7;
   FP_PARM.AI2_Max := 100.0;
   FP_PARM.AI3_Max := 100.0;
   FP_PARM.AO1a_Max := 100.0;
   FP_PARM.AO2a_Max := 100.0;
   FP_PARM.AO3a_Max := 100.0;
   FP_PARM.AO1b_Max := 10.7;
   FP_PARM.AO2b_Max := 5.5;
   FP_PARM.AO3b_Max := 100.0;
   SEL := FALSE;
   MD := FALSE;
   BUSF := FALSE;
   DOPR := FALSE;
   DTEST := TRUE;
   SFS := FALSE;
   ES := TRUE;
   INTL.OK := TRUE;
   INTL_SEQ_STR1.OK := TRUE;
   INTL_SEQ_STR2.OK := TRUE;
   INTL_SEQ_STP.OK := TRUE;
   LAMP1 := TRUE;
   LAMP2 := TRUE;
   MAN := TRUE;
   MSW.EXT.ModeBit2 := TRUE;
   MSW.EXT.AlarmPresent := TRUE;
   MSW.EXT.AlarmFailUnAck := TRUE;
   MSW.Status := 201;
   MSW.TimeStamp := 16#12F0;
   BlockInfo.Ace_Version := 80;
   BlockInfo.Ace_BuildNo := 13;
   BlockInfo.State_Act := 607;
   BlockInfo.State_Prev := 405;
   BlockInfo.DB_Number := 4416;
   FP_CMD.Manual := TRUE;
   FP_EN.PB_QStop := TRUE;
   FP_DIM.Auto := TRUE;
   FP_DIM.Local := TRUE;
   FP_DIM.Reset := TRUE;
   FP_SHOW.PB_Auto := TRUE;
   FP_SHOW.PB_Local := TRUE;
   FP_SHOW.PB_Manual := TRUE;
   FP_SHOW.PB_Start1 := TRUE;
   FP_SHOW.PB_Stop := TRUE;
   FP_SHOW.AI1 := TRUE;
   FP_SHOW.AI2 := TRUE;
   FP_SHOW.AI3 := TRUE;
   FP_SHOW.SP := TRUE;
   FP_SHOW.OVL := TRUE;
   FP_SHOW.SSW := TRUE;
   FP_SHOW.STALL := TRUE;
   FP_SHOW.EARTH := TRUE;
   FP_SHOW.UBAL := TRUE;
   FP_SHOW.GFA := TRUE;
   FP_SHOW.GWA := TRUE;
   FP_SHOW.BUSF := TRUE;
   FP_SHOW.DOPR := TRUE;
   FP_SHOW.DTEST := TRUE;
   FP_SHOW.LSTR1 := TRUE;
   FP_PARM.StartWarn_Acc := 15;
   FP_PARM.RunDelay1_Acc := 5;
   FP_PARM.DelayStop_Acc := 5;
   FP_PARM.ReturnMon_Acc := 2;
   FP_PARM.MD_Freq_SP := 1;
   FP_PARM.StopReason := 11;
   FP_PARM.INTL := TRUE;
   FP_PARM.INTL_SEQ_STR1 := TRUE;
   FP_PARM.INTL_SEQ_STR2 := TRUE;
   FP_PARM.INTL_SEQ_STP := TRUE;
   FP_SIM.OVL_Enable := TRUE;
   FP_SIM.RDY_Enable := TRUE;
   FP_SIM.SSW_Enable := TRUE;
   FP_SIM.TFA_Enable := TRUE;
   FP_SIM.MCC_Enable := TRUE;
   FP_SIM.DRDY_Enable := TRUE;
   FP_SIM.MD_Enable := TRUE;
   FP_SIM.GFA_Enable := TRUE;
   FP_SIM.GWA_Enable := TRUE;
   FP_SIM.STALL_Enable := TRUE;
   FP_SIM.EARTH_Enable := TRUE;
   FP_SIM.UBAL_Enable := TRUE;
   FP_SIM.BUSF_Enable := TRUE;
   FP_SIM.RET1_Enable := TRUE;
   FP_SIM.RET2_Enable := TRUE;
   FP_SIM.DOPR_Enable := TRUE;
   FP_SIM.ACK_Enable := TRUE;
   FP_SIM.LSTP_Enable := TRUE;
   FP_SIM.REM_Enable := TRUE;
   FP_SIM.SFS_Enable := TRUE;
   FP_SIM.SLS_Enable := TRUE;
   FP_SIM.ES_Enable := TRUE;
   FP_SIM.WORK.Flash_Slow := TRUE;
   AdapterBlock.Intell_Type := 282;
   AdapterBlock.VersionNo := 220;
   AdapterBlock.FuncType := 41;
   AdapterBlock.Options := 1;
   AdapterBlock.NetNo := 106;
   AdapterBlock.NodeNo := 76;
   AdapterBlock.Flash_Slow := TRUE;
   AdapterBlock.Flash_Fast := TRUE;
   AdapterBlock.MAN := TRUE;
   AdapterBlock.HMI_INT[11] := 6;
   AdapterBlock.HMI_REAL[9] := 100.0;
   AdapterBlock.HMI_REAL[10] := 100.0;
   AdapterBlock.HMI_REAL[12] := 100.0;
   AdapterBlock.HMI_BOOL[34] := TRUE;
   AdapterBlock.HMI_BOOL[35] := TRUE;
   AdapterBlock.HMI_BOOL[65] := TRUE;
   AdapterBlock.HMI_BOOL[89] := TRUE;
   STATE.Alarm := TRUE;
   ONS.Unimotor := TRUE;
   ONS.MD_OnOff := TRUE;
   ONS.Cmd_Manual := TRUE;
   ONS.GLTP := TRUE;
   ONS.CMD_Start1 := TRUE;
   ONS.CMD_Start2 := TRUE;
   ONS.SecPulse1 := TRUE;
   StatusWork := 201;
   ModePointer := 52;
   AlarmNo := 23;
   AlarmNo_Old := 23;
   StartWarn_Mem := 15;
   RunDelay1_Mem := 5;
   DelayStop_Mem := 5;
   ReturnMon_Mem := 2;
   ModeManual := TRUE;
   FromStopState := TRUE;
   ALARM_AlarmPresent := TRUE;
   ChangeDir1_Done := TRUE;
   ChangeDir2_Done := TRUE;
   OUT.LAMP1 := TRUE;
   OUT.LAMP2 := TRUE;
   OUT.MAN := TRUE;
   OUT.INTL_OK_STAT := TRUE;
   OUT.INTL_SEQ_STR1_OK_STAT := TRUE;
   OUT.INTL_SEQ_STR2_OK_STAT := TRUE;
   OUT.INTL_SEQ_STP_OK_STAT := TRUE;
   MSW_Status_Trans := 201;
END_DATA_BLOCK

